LIN {X 0,Y 453.144,Z 723.625,A -85,B 0,C 180,E1 16875.324,E2 16875.324} C_VEL
LIN {X 0,Y 454.014,Z 710.614,A -85,B 0,C 180,E1 16875.765,E2 16875.765} C_VEL
LIN {X 0,Y 429.058,Z 654.338,A -85,B 0,C 180,E1 16879.298,E2 16879.298} C_VEL
LIN {X 0,Y 404.681,Z 601.31,A -85,B 0,C 180,E1 16882.971,E2 16882.971} C_VEL
LIN {X 0,Y 404.836,Z 601.31,A -85,B 0,C 180,E1 16889.422,E2 16889.422} C_VEL
LIN {X 0,Y 405.105,Z 601.31,A -85,B 0,C 180,E1 16895.708,E2 16895.708} C_VEL
LIN {X 0,Y 405.45,Z 601.31,A -85,B 0,C 180,E1 16902.605,E2 16902.605} C_VEL
LIN {X 0,Y 405.795,Z 601.31,A -85,B 0,C 180,E1 16909.24,E2 16909.24} C_VEL
LIN {X 0,Y 406.34,Z 601.31,A -85,B 0,C 180,E1 16915.721,E2 16915.721} C_VEL
LIN {X 0,Y 406.534,Z 601.31,A -85,B 0,C 180,E1 16922.133,E2 16922.133} C_VEL
LIN {X 0,Y 405.998,Z 601.31,A -85,B 0,C 180,E1 16928.581,E2 16928.581} C_VEL
LIN {X 0,Y 405.598,Z 601.31,A -85,B 0,C 180,E1 16935.153,E2 16935.153} C_VEL
LIN {X 0,Y 405.276,Z 601.31,A -85,B 0,C 180,E1 16941.947,E2 16941.947} C_VEL
LIN {X 0,Y 404.862,Z 601.31,A -85,B 0,C 180,E1 16949.103,E2 16949.103} C_VEL
LIN {X 0,Y 404.667,Z 601.31,A -85,B 0,C 180,E1 16954.527,E2 16954.527} C_VEL
LIN {X 0,Y 404.635,Z 601.31,A -85,B 0,C 180,E1 16961.494,E2 16961.494} C_VEL
LIN {X 0,Y 404.616,Z 601.411,A -85,B 0,C 180,E1 16963.759,E2 16963.759} C_VEL
LIN {X 0,Y 407.142,Z 607.04,A -85,B 0,C 180,E1 16964.41,E2 16964.41} C_VEL
LIN {X 0,Y 426.451,Z 643.441,A -85,B 0,C 180,E1 16968.623,E2 16968.623} C_VEL
LIN {X 0,Y 441.542,Z 679.841,A -85,B 0,C 180,E1 16971.916,E2 16971.916} C_VEL
LIN {X 0,Y 445.49,Z 694.589,A -85,B 0,C 180,E1 16973.129,E2 16973.129} C_VEL
LIN {X 0,Y 440.363,Z 731.801,A -85,B 0,C 180,E1 16975.298,E2 16975.298} C_VEL
LIN {X 0,Y 433.881,Z 767.453,A -85,B 0,C 180,E1 16978.257,E2 16978.257} C_VEL
LIN {X 0,Y 426.951,Z 799.424,A -85,B 0,C 180,E1 16981.945,E2 16981.945} C_VEL
LIN {X 0,Y 420.677,Z 825.936,A -85,B 0,C 180,E1 16986.09,E2 16986.09} C_VEL
LIN {X 0,Y 415.363,Z 848.097,A -85,B 0,C 180,E1 16990.828,E2 16990.828} C_VEL
LIN {X 0,Y 411.855,Z 864.058,A -85,B 0,C 180,E1 16995.615,E2 16995.615} C_VEL
LIN {X 0,Y 409.78,Z 874.937,A -85,B 0,C 180,E1 17000.416,E2 17000.416} C_VEL
LIN {X 0,Y 408.702,Z 881.698,A -85,B 0,C 180,E1 17005.742,E2 17005.742} C_VEL
LIN {X 0,Y 408.585,Z 883.379,A -85,B 0,C 180,E1 17009.994,E2 17009.994} C_VEL
LIN {X 0,Y 408.851,Z 880.711,A -85,B 0,C 180,E1 17015.31,E2 17015.31} C_VEL
LIN {X 0,Y 410.092,Z 872.747,A -85,B 0,C 180,E1 17020.64,E2 17020.64} C_VEL
LIN {X 0,Y 412.907,Z 859.065,A -85,B 0,C 180,E1 17025.969,E2 17025.969} C_VEL
LIN {X 0,Y 417.3,Z 839.904,A -85,B 0,C 180,E1 17031.006,E2 17031.006} C_VEL
LIN {X 0,Y 423.261,Z 814.998,A -85,B 0,C 180,E1 17035.669,E2 17035.669} C_VEL
LIN {X 0,Y 430.079,Z 785.455,A -85,B 0,C 180,E1 17039.706,E2 17039.706} C_VEL
LIN {X 0,Y 436.704,Z 752.798,A -85,B 0,C 180,E1 17042.97,E2 17042.97} C_VEL
LIN {X 0,Y 442.585,Z 716.698,A -85,B 0,C 180,E1 17045.585,E2 17045.585} C_VEL
LIN {X 0,Y 445.078,Z 692.222,A -85,B 0,C 180,E1 17046.937,E2 17046.937} C_VEL
LIN {X 0,Y 433.84,Z 659.714,A -85,B 0,C 180,E1 17049.714,E2 17049.714} C_VEL
LIN {X 0,Y 416.42,Z 623.579,A -85,B 0,C 180,E1 17053.415,E2 17053.415} C_VEL
LIN {X 0,Y 404.643,Z 601.978,A -85,B 0,C 180,E1 17056.084,E2 17056.084} C_VEL
LIN {X 0,Y 404.565,Z 601.31,A -85,B 0,C 180,E1 17061.851,E2 17061.851} C_VEL
LIN {X 0,Y 404.943,Z 601.976,A -85,B 0,C 180,E1 17068.085,E2 17068.085} C_VEL
LIN {X 0,Y 427.922,Z 668.698,A -85,B 0,C 180,E1 17071.46,E2 17071.46} C_VEL
LIN {X 0,Y 428.67,Z 678.715,A -85,B 0,C 180,E1 17071.781,E2 17071.781} C_VEL
LIN {X 0,Y 425.713,Z 719.893,A -85,B 0,C 180,E1 17073.236,E2 17073.236} C_VEL
LIN {X 0,Y 421.872,Z 759.16,A -85,B 0,C 180,E1 17075.471,E2 17075.471} C_VEL
LIN {X 0,Y 417.99,Z 794.434,A -85,B 0,C 180,E1 17078.39,E2 17078.39} C_VEL
LIN {X 0,Y 414.582,Z 824.543,A -85,B 0,C 180,E1 17081.831,E2 17081.831} C_VEL
LIN {X 0,Y 411.814,Z 848.973,A -85,B 0,C 180,E1 17085.626,E2 17085.626} C_VEL
LIN {X 0,Y 410.114,Z 868.93,A -85,B 0,C 180,E1 17089.898,E2 17089.898} C_VEL
LIN {X 0,Y 409.272,Z 882.602,A -85,B 0,C 180,E1 17094.161,E2 17094.161} C_VEL
LIN {X 0,Y 409.19,Z 891.235,A -85,B 0,C 180,E1 17098.574,E2 17098.574} C_VEL
LIN {X 0,Y 409.569,Z 894.347,A -85,B 0,C 180,E1 17102.122,E2 17102.122} C_VEL
LIN {X 0,Y 411.139,Z 893.587,A -85,B 0,C 180,E1 17106.349,E2 17106.349} C_VEL
LIN {X 0,Y 413.508,Z 887.959,A -85,B 0,C 180,E1 17110.557,E2 17110.557} C_VEL
LIN {X 0,Y 417.618,Z 875.892,A -85,B 0,C 180,E1 17115.115,E2 17115.115} C_VEL
LIN {X 0,Y 422.993,Z 858.13,A -85,B 0,C 180,E1 17119.349,E2 17119.349} C_VEL
LIN {X 0,Y 430.431,Z 833.334,A -85,B 0,C 180,E1 17123.442,E2 17123.442} C_VEL
LIN {X 0,Y 439.545,Z 802.14,A -85,B 0,C 180,E1 17127.174,E2 17127.174} C_VEL
LIN {X 0,Y 450.951,Z 763.363,A -85,B 0,C 180,E1 17130.54,E2 17130.54} C_VEL
LIN {X 0,Y 462.959,Z 721.781,A -85,B 0,C 180,E1 17133.048,E2 17133.048} C_VEL
LIN {X 0,Y 469.674,Z 695.489,A -85,B 0,C 180,E1 17134.267,E2 17134.267} C_VEL
LIN {X 0,Y 469.832,Z 688.161,A -85,B 0,C 180,E1 17136.141,E2 17136.141} C_VEL
LIN {X 0,Y 470.531,Z 686.318,A -85,B 0,C 180,E1 17137.657,E2 17137.657} C_VEL
LIN {X 0,Y 471.824,Z 691.946,A -85,B 0,C 180,E1 17139.617,E2 17139.617} C_VEL
LIN {X 0,Y 472.889,Z 702.024,A -85,B 0,C 180,E1 17141.096,E2 17141.096} C_VEL
LIN {X 0,Y 472.481,Z 713.92,A -85,B 0,C 180,E1 17142.03,E2 17142.03} C_VEL
LIN {X 0,Y 462.296,Z 759.297,A -85,B 0,C 180,E1 17143.95,E2 17143.95} C_VEL
LIN {X 0,Y 450.752,Z 803.897,A -85,B 0,C 180,E1 17146.773,E2 17146.773} C_VEL
LIN {X 0,Y 438.988,Z 845.741,A -85,B 0,C 180,E1 17150.484,E2 17150.484} C_VEL
LIN {X 0,Y 428.197,Z 882.986,A -85,B 0,C 180,E1 17154.933,E2 17154.933} C_VEL
LIN {X 0,Y 419.612,Z 914.659,A -85,B 0,C 180,E1 17159.961,E2 17159.961} C_VEL
LIN {X 0,Y 413.13,Z 941.761,A -85,B 0,C 180,E1 17165.638,E2 17165.638} C_VEL
LIN {X 0,Y 409.271,Z 963.039,A -85,B 0,C 180,E1 17171.664,E2 17171.664} C_VEL
LIN {X 0,Y 407.76,Z 977.862,A -85,B 0,C 180,E1 17177.669,E2 17177.669} C_VEL
LIN {X 0,Y 407.499,Z 985.661,A -85,B 0,C 180,E1 17182.528,E2 17182.528} C_VEL
LIN {X 0,Y 407.719,Z 989.763,A -85,B 0,C 180,E1 17187.876,E2 17187.876} C_VEL
LIN {X 0,Y 407.669,Z 989.715,A -85,B 0,C 180,E1 17192.136,E2 17192.136} C_VEL
LIN {X 0,Y 407.522,Z 985.383,A -85,B 0,C 180,E1 17197.483,E2 17197.483} C_VEL
LIN {X 0,Y 407.925,Z 976.144,A -85,B 0,C 180,E1 17202.883,E2 17202.883} C_VEL
LIN {X 0,Y 409.066,Z 963.513,A -85,B 0,C 180,E1 17207.72,E2 17207.72} C_VEL
LIN {X 0,Y 406.112,Z 956.241,A -85,B 0,C 180,E1 17209.923,E2 17209.923} C_VEL
LIN {X 0,Y 403.464,Z 948.232,A -85,B 0,C 180,E1 17212.111,E2 17212.111} C_VEL
LIN {X 0,Y 408.092,Z 924.272,A -85,B 0,C 180,E1 17217.467,E2 17217.467} C_VEL
LIN {X 0,Y 414.359,Z 895.799,A -85,B 0,C 180,E1 17222.261,E2 17222.261} C_VEL
LIN {X 0,Y 421.833,Z 862.647,A -85,B 0,C 180,E1 17226.508,E2 17226.508} C_VEL
LIN {X 0,Y 430.114,Z 823.849,A -85,B 0,C 180,E1 17230.223,E2 17230.223} C_VEL
LIN {X 0,Y 437.983,Z 781.87,A -85,B 0,C 180,E1 17233.15,E2 17233.15} C_VEL
LIN {X 0,Y 444.627,Z 738.33,A -85,B 0,C 180,E1 17235.268,E2 17235.268} C_VEL
LIN {X 0,Y 446.908,Z 712.636,A -85,B 0,C 180,E1 17236.208,E2 17236.208} C_VEL
LIN {X 0,Y 424.33,Z 661.374,A -85,B 0,C 180,E1 17239.508,E2 17239.508} C_VEL
LIN {X 0,Y 396.721,Z 601.31,A -85,B 0,C 180,E1 17243.82,E2 17243.82} C_VEL
LIN {X 0,Y 396.924,Z 601.31,A -85,B 0,C 180,E1 17250.251,E2 17250.251} C_VEL
LIN {X 0,Y 397.264,Z 601.31,A -85,B 0,C 180,E1 17257.581,E2 17257.581} C_VEL
LIN {X 0,Y 397.599,Z 601.31,A -85,B 0,C 180,E1 17264.529,E2 17264.529} C_VEL
LIN {X 0,Y 398.087,Z 601.31,A -85,B 0,C 180,E1 17271.778,E2 17271.778} C_VEL
LIN {X 0,Y 398.566,Z 601.31,A -85,B 0,C 180,E1 17277.819,E2 17277.819} C_VEL
LIN {X 0,Y 398.622,Z 601.31,A -85,B 0,C 180,E1 17282.175,E2 17282.175} C_VEL
LIN {X 0,Y 398.065,Z 601.31,A -85,B 0,C 180,E1 17288.753,E2 17288.753} C_VEL
LIN {X 0,Y 397.646,Z 601.31,A -85,B 0,C 180,E1 17295.464,E2 17295.464} C_VEL
LIN {X 0,Y 397.287,Z 601.31,A -85,B 0,C 180,E1 17302.412,E2 17302.412} C_VEL
LIN {X 0,Y 396.937,Z 601.31,A -85,B 0,C 180,E1 17309.741,E2 17309.741} C_VEL
LIN {X 0,Y 396.708,Z 601.31,A -85,B 0,C 180,E1 17316.66,E2 17316.66} C_VEL
LIN {X 0,Y 396.735,Z 601.61,A -85,B 0,C 180,E1 17322.493,E2 17322.493} C_VEL
LIN {X 0,Y 399.282,Z 607.13,A -85,B 0,C 180,E1 17323.171,E2 17323.171} C_VEL
LIN {X 0,Y 417.822,Z 641.308,A -85,B 0,C 180,E1 17327.427,E2 17327.427} C_VEL
LIN {X 0,Y 433.732,Z 678.097,A -85,B 0,C 180,E1 17330.964,E2 17330.964} C_VEL
LIN {X 0,Y 439.018,Z 697.43,A -85,B 0,C 180,E1 17332.614,E2 17332.614} C_VEL
LIN {X 0,Y 433.748,Z 733.916,A -85,B 0,C 180,E1 17334.796,E2 17334.796} C_VEL
LIN {X 0,Y 426.94,Z 769.727,A -85,B 0,C 180,E1 17337.829,E2 17337.829} C_VEL
LIN {X 0,Y 420.013,Z 800.415,A -85,B 0,C 180,E1 17341.439,E2 17341.439} C_VEL
LIN {X 0,Y 413.497,Z 826.928,A -85,B 0,C 180,E1 17345.648,E2 17345.648} C_VEL
LIN {X 0,Y 407.947,Z 849.099,A -85,B 0,C 180,E1 17350.465,E2 17350.465} C_VEL
LIN {X 0,Y 404.23,Z 865.06,A -85,B 0,C 180,E1 17355.338,E2 17355.338} C_VEL
LIN {X 0,Y 402.037,Z 875.93,A -85,B 0,C 180,E1 17360.23,E2 17360.23} C_VEL
LIN {X 0,Y 400.887,Z 882.687,A -85,B 0,C 180,E1 17365.659,E2 17365.659} C_VEL
LIN {X 0,Y 400.763,Z 884.365,A -85,B 0,C 180,E1 17369.994,E2 17369.994} C_VEL
LIN {X 0,Y 401.035,Z 881.701,A -85,B 0,C 180,E1 17375.414,E2 17375.414} C_VEL
LIN {X 0,Y 402.381,Z 873.742,A -85,B 0,C 180,E1 17380.846,E2 17380.846} C_VEL
LIN {X 0,Y 405.349,Z 860.066,A -85,B 0,C 180,E1 17386.275,E2 17386.275} C_VEL
LIN {X 0,Y 409.947,Z 840.904,A -85,B 0,C 180,E1 17391.401,E2 17391.401} C_VEL
LIN {X 0,Y 416.115,Z 816.225,A -85,B 0,C 180,E1 17396.102,E2 17396.102} C_VEL
LIN {X 0,Y 422.995,Z 787.652,A -85,B 0,C 180,E1 17400.092,E2 17400.092} C_VEL
LIN {X 0,Y 429.834,Z 755.218,A -85,B 0,C 180,E1 17403.415,E2 17403.415} C_VEL
LIN {X 0,Y 435.998,Z 719.092,A -85,B 0,C 180,E1 17406.095,E2 17406.095} C_VEL
LIN {X 0,Y 438.752,Z 695.217,A -85,B 0,C 180,E1 17407.432,E2 17407.432} C_VEL
LIN {X 0,Y 428.14,Z 663.804,A -85,B 0,C 180,E1 17410.203,E2 17410.203} C_VEL
LIN {X 0,Y 411.375,Z 628.716,A -85,B 0,C 180,E1 17413.89,E2 17413.89} C_VEL
LIN {X 0,Y 396.772,Z 602.597,A -85,B 0,C 180,E1 17417.323,E2 17417.323} C_VEL
LIN {X 0,Y 396.68,Z 601.31,A -85,B 0,C 180,E1 17417.552,E2 17417.552} C_VEL
LIN {X 0,Y 396.704,Z 601.31,A -85,B 0,C 180,E1 17425.058,E2 17425.058} C_VEL
LIN {X 0,Y 396.951,Z 601.31,A -85,B 0,C 180,E1 17427.466,E2 17427.466} C_VEL
LIN {X 0,Y 420.826,Z 670.997,A -85,B 0,C 180,E1 17431.112,E2 17431.112} C_VEL
LIN {X 0,Y 420.941,Z 686.929,A -85,B 0,C 180,E1 17431.596,E2 17431.596} C_VEL
LIN {X 0,Y 417.659,Z 727.911,A -85,B 0,C 180,E1 17433.231,E2 17433.231} C_VEL
LIN {X 0,Y 413.648,Z 766.912,A -85,B 0,C 180,E1 17435.672,E2 17435.672} C_VEL
LIN {X 0,Y 409.558,Z 802.307,A -85,B 0,C 180,E1 17438.864,E2 17438.864} C_VEL
LIN {X 0,Y 406.016,Z 832.346,A -85,B 0,C 180,E1 17442.636,E2 17442.636} C_VEL
LIN {X 0,Y 403.418,Z 856.03,A -85,B 0,C 180,E1 17446.706,E2 17446.706} C_VEL
LIN {X 0,Y 401.855,Z 875.142,A -85,B 0,C 180,E1 17451.33,E2 17451.33} C_VEL
LIN {X 0,Y 401.38,Z 887.036,A -85,B 0,C 180,E1 17455.674,E2 17455.674} C_VEL
LIN {X 0,Y 401.482,Z 893.849,A -85,B 0,C 180,E1 17460.003,E2 17460.003} C_VEL
LIN {X 0,Y 402.47,Z 895.827,A -85,B 0,C 180,E1 17464.32,E2 17464.32} C_VEL
LIN {X 0,Y 404.529,Z 892.945,A -85,B 0,C 180,E1 17468.618,E2 17468.618} C_VEL
LIN {X 0,Y 408.246,Z 883.721,A -85,B 0,C 180,E1 17473.413,E2 17473.413} C_VEL
LIN {X 0,Y 412.904,Z 870.089,A -85,B 0,C 180,E1 17477.566,E2 17477.566} C_VEL
LIN {X 0,Y 419.579,Z 850.051,A -85,B 0,C 180,E1 17481.723,E2 17481.723} C_VEL
LIN {X 0,Y 428.729,Z 821.406,A -85,B 0,C 180,E1 17485.932,E2 17485.932} C_VEL
LIN {X 0,Y 440.153,Z 786.19,A -85,B 0,C 180,E1 17489.656,E2 17489.656} C_VEL
LIN {X 0,Y 452.998,Z 746.965,A -85,B 0,C 180,E1 17492.635,E2 17492.635} C_VEL
LIN {X 0,Y 465.569,Z 706.07,A -85,B 0,C 180,E1 17494.732,E2 17494.732} C_VEL
LIN {X 0,Y 467.104,Z 699.977,A -85,B 0,C 180,E1 17495.095,E2 17495.095} C_VEL
LIN {X 0,Y 467.92,Z 694.621,A -85,B 0,C 180,E1 17496.923,E2 17496.923} C_VEL
LIN {X 0,Y 468.515,Z 695.099,A -85,B 0,C 180,E1 17498.092,E2 17498.092} C_VEL
LIN {X 0,Y 469.391,Z 701.137,A -85,B 0,C 180,E1 17499.712,E2 17499.712} C_VEL
LIN {X 0,Y 469.233,Z 712.69,A -85,B 0,C 180,E1 17500.993,E2 17500.993} C_VEL
LIN {X 0,Y 456.969,Z 763.857,A -85,B 0,C 180,E1 17503.339,E2 17503.339} C_VEL
LIN {X 0,Y 444.904,Z 806.362,A -85,B 0,C 180,E1 17506.155,E2 17506.155} C_VEL
LIN {X 0,Y 432.505,Z 847.465,A -85,B 0,C 180,E1 17509.936,E2 17509.936} C_VEL
LIN {X 0,Y 421.413,Z 883.423,A -85,B 0,C 180,E1 17514.373,E2 17514.373} C_VEL
LIN {X 0,Y 412.458,Z 914.186,A -85,B 0,C 180,E1 17519.385,E2 17519.385} C_VEL
LIN {X 0,Y 405.947,Z 939.975,A -85,B 0,C 180,E1 17524.883,E2 17524.883} C_VEL
LIN {X 0,Y 401.699,Z 961.213,A -85,B 0,C 180,E1 17530.941,E2 17530.941} C_VEL
LIN {X 0,Y 399.921,Z 977.012,A -85,B 0,C 180,E1 17537.423,E2 17537.423} C_VEL
LIN {X 0,Y 399.618,Z 984.745,A -85,B 0,C 180,E1 17542.38,E2 17542.38} C_VEL
LIN {X 0,Y 399.888,Z 988.813,A -85,B 0,C 180,E1 17547.834,E2 17547.834} C_VEL
LIN {X 0,Y 399.842,Z 988.709,A -85,B 0,C 180,E1 17552.178,E2 17552.178} C_VEL
LIN {X 0,Y 399.685,Z 984.293,A -85,B 0,C 180,E1 17557.631,E2 17557.631} C_VEL
LIN {X 0,Y 400.089,Z 974.873,A -85,B 0,C 180,E1 17563.14,E2 17563.14} C_VEL
LIN {X 0,Y 401.48,Z 960.573,A -85,B 0,C 180,E1 17568.582,E2 17568.582} C_VEL
LIN {X 0,Y 403.464,Z 948.232,A -85,B 0,C 180,E1 17572.111,E2 17572.111} C_VEL
LIN {X 0,Y 401.121,Z 939.612,A -85,B 0,C 180,E1 17574.259,E2 17574.259} C_VEL
LIN {X 0,Y 399.038,Z 930.299,A -85,B 0,C 180,E1 17576.378,E2 17576.378} C_VEL
LIN {X 0,Y 405.037,Z 903.022,A -85,B 0,C 180,E1 17581.397,E2 17581.397} C_VEL
LIN {X 0,Y 412.444,Z 871.136,A -85,B 0,C 180,E1 17585.845,E2 17585.845} C_VEL
LIN {X 0,Y 420.387,Z 835.553,A -85,B 0,C 180,E1 17589.607,E2 17589.607} C_VEL
LIN {X 0,Y 428.414,Z 796.139,A -85,B 0,C 180,E1 17592.707,E2 17592.707} C_VEL
LIN {X 0,Y 435.678,Z 753.012,A -85,B 0,C 180,E1 17595.129,E2 17595.129} C_VEL
LIN {X 0,Y 439.896,Z 715.013,A -85,B 0,C 180,E1 17596.636,E2 17596.636} C_VEL
LIN {X 0,Y 419.655,Z 668.36,A -85,B 0,C 180,E1 17599.719,E2 17599.719} C_VEL
LIN {X 0,Y 388.811,Z 601.31,A -85,B 0,C 180,E1 17604.558,E2 17604.558} C_VEL
LIN {X 0,Y 389.049,Z 601.31,A -85,B 0,C 180,E1 17612.14,E2 17612.14} C_VEL
LIN {X 0,Y 389.433,Z 601.31,A -85,B 0,C 180,E1 17619.504,E2 17619.504} C_VEL
LIN {X 0,Y 389.826,Z 601.31,A -85,B 0,C 180,E1 17626.514,E2 17626.514} C_VEL
LIN {X 0,Y 390.335,Z 601.31,A -85,B 0,C 180,E1 17633.311,E2 17633.311} C_VEL
LIN {X 0,Y 390.868,Z 601.31,A -85,B 0,C 180,E1 17639.997,E2 17639.997} C_VEL
LIN {X 0,Y 390.34,Z 601.31,A -85,B 0,C 180,E1 17646.683,E2 17646.683} C_VEL
LIN {X 0,Y 389.843,Z 601.31,A -85,B 0,C 180,E1 17653.643,E2 17653.643} C_VEL
LIN {X 0,Y 389.412,Z 601.31,A -85,B 0,C 180,E1 17660.941,E2 17660.941} C_VEL
LIN {X 0,Y 389.034,Z 601.31,A -85,B 0,C 180,E1 17667.854,E2 17667.854} C_VEL
LIN {X 0,Y 388.844,Z 601.31,A -85,B 0,C 180,E1 17675.074,E2 17675.074} C_VEL
LIN {X 0,Y 388.797,Z 601.546,A -85,B 0,C 180,E1 17681.118,E2 17681.118} C_VEL
LIN {X 0,Y 391.283,Z 607.066,A -85,B 0,C 180,E1 17681.818,E2 17681.818} C_VEL
LIN {X 0,Y 409.624,Z 639.903,A -85,B 0,C 180,E1 17686.242,E2 17686.242} C_VEL
LIN {X 0,Y 426.017,Z 676.952,A -85,B 0,C 180,E1 17690.025,E2 17690.025} C_VEL
LIN {X 0,Y 432.632,Z 699.526,A -85,B 0,C 180,E1 17692.046,E2 17692.046} C_VEL
LIN {X 0,Y 427.133,Z 736.226,A -85,B 0,C 180,E1 17694.293,E2 17694.293} C_VEL
LIN {X 0,Y 420.051,Z 771.896,A -85,B 0,C 180,E1 17697.381,E2 17697.381} C_VEL
LIN {X 0,Y 412.682,Z 803.295,A -85,B 0,C 180,E1 17701.184,E2 17701.184} C_VEL
LIN {X 0,Y 405.602,Z 830.769,A -85,B 0,C 180,E1 17705.731,E2 17705.731} C_VEL
LIN {X 0,Y 400.01,Z 852,A -85,B 0,C 180,E1 17710.601,E2 17710.601} C_VEL
LIN {X 0,Y 395.958,Z 868.944,A -85,B 0,C 180,E1 17716.156,E2 17716.156} C_VEL
LIN {X 0,Y 393.908,Z 878.753,A -85,B 0,C 180,E1 17721.143,E2 17721.143} C_VEL
LIN {X 0,Y 393.089,Z 883.674,A -85,B 0,C 180,E1 17725.572,E2 17725.572} C_VEL
LIN {X 0,Y 392.955,Z 885.35,A -85,B 0,C 180,E1 17729.994,E2 17729.994} C_VEL
LIN {X 0,Y 393.241,Z 882.688,A -85,B 0,C 180,E1 17735.522,E2 17735.522} C_VEL
LIN {X 0,Y 394.681,Z 874.735,A -85,B 0,C 180,E1 17741.061,E2 17741.061} C_VEL
LIN {X 0,Y 397.776,Z 861.078,A -85,B 0,C 180,E1 17746.594,E2 17746.594} C_VEL
LIN {X 0,Y 402.63,Z 841.907,A -85,B 0,C 180,E1 17751.809,E2 17751.809} C_VEL
LIN {X 0,Y 409.074,Z 817.24,A -85,B 0,C 180,E1 17756.585,E2 17756.585} C_VEL
LIN {X 0,Y 416.212,Z 788.636,A -85,B 0,C 180,E1 17760.635,E2 17760.635} C_VEL
LIN {X 0,Y 423.326,Z 756.172,A -85,B 0,C 180,E1 17763.998,E2 17763.998} C_VEL
LIN {X 0,Y 429.751,Z 719.457,A -85,B 0,C 180,E1 17766.741,E2 17766.741} C_VEL
LIN {X 0,Y 432.249,Z 697.341,A -85,B 0,C 180,E1 17768.015,E2 17768.015} C_VEL
LIN {X 0,Y 421.482,Z 665.442,A -85,B 0,C 180,E1 17770.935,E2 17770.935} C_VEL
LIN {X 0,Y 404.201,Z 629.523,A -85,B 0,C 180,E1 17774.901,E2 17774.901} C_VEL
LIN {X 0,Y 390.003,Z 605.572,A -85,B 0,C 180,E1 17778.345,E2 17778.345} C_VEL
LIN {X 0,Y 388.737,Z 601.31,A -85,B 0,C 180,E1 17778.808,E2 17778.808} C_VEL
LIN {X 0,Y 388.985,Z 601.31,A -85,B 0,C 180,E1 17786.898,E2 17786.898} C_VEL
LIN {X 0,Y 412.526,Z 669.642,A -85,B 0,C 180,E1 17790.575,E2 17790.575} C_VEL
LIN {X 0,Y 414.213,Z 677.972,A -85,B 0,C 180,E1 17790.919,E2 17790.919} C_VEL
LIN {X 0,Y 411.094,Z 719.632,A -85,B 0,C 180,E1 17792.43,E2 17792.43} C_VEL
LIN {X 0,Y 407.087,Z 758.185,A -85,B 0,C 180,E1 17794.666,E2 17794.666} C_VEL
LIN {X 0,Y 402.859,Z 794.573,A -85,B 0,C 180,E1 17797.74,E2 17797.74} C_VEL
LIN {X 0,Y 399.041,Z 826.575,A -85,B 0,C 180,E1 17801.517,E2 17801.517} C_VEL
LIN {X 0,Y 396.091,Z 851.835,A -85,B 0,C 180,E1 17805.608,E2 17805.608} C_VEL
LIN {X 0,Y 394.356,Z 871.599,A -85,B 0,C 180,E1 17810.048,E2 17810.048} C_VEL
LIN {X 0,Y 393.543,Z 885.173,A -85,B 0,C 180,E1 17814.48,E2 17814.48} C_VEL
LIN {X 0,Y 393.556,Z 893.492,A -85,B 0,C 180,E1 17818.9,E2 17818.9} C_VEL
LIN {X 0,Y 393.94,Z 896.554,A -85,B 0,C 180,E1 17822.207,E2 17822.207} C_VEL
LIN {X 0,Y 395.687,Z 896.345,A -85,B 0,C 180,E1 17826.598,E2 17826.598} C_VEL
LIN {X 0,Y 398.826,Z 890.34,A -85,B 0,C 180,E1 17831.505,E2 17831.505} C_VEL
LIN {X 0,Y 403.433,Z 878.844,A -85,B 0,C 180,E1 17836.082,E2 17836.082} C_VEL
LIN {X 0,Y 409.889,Z 861.011,A -85,B 0,C 180,E1 17840.558,E2 17840.558} C_VEL
LIN {X 0,Y 418.813,Z 835.899,A -85,B 0,C 180,E1 17844.927,E2 17844.927} C_VEL
LIN {X 0,Y 430.242,Z 803.687,A -85,B 0,C 180,E1 17848.959,E2 17848.959} C_VEL
LIN {X 0,Y 444.537,Z 764.527,A -85,B 0,C 180,E1 17852.464,E2 17852.464} C_VEL
LIN {X 0,Y 458.962,Z 723.662,A -85,B 0,C 180,E1 17854.961,E2 17854.961} C_VEL
LIN {X 0,Y 464.376,Z 706.896,A -85,B 0,C 180,E1 17855.698,E2 17855.698} C_VEL
LIN {X 0,Y 465.29,Z 703.344,A -85,B 0,C 180,E1 17856.422,E2 17856.422} C_VEL
LIN {X 0,Y 466.118,Z 702.017,A -85,B 0,C 180,E1 17857.685,E2 17857.685} C_VEL
LIN {X 0,Y 466.541,Z 706.311,A -85,B 0,C 180,E1 17859.045,E2 17859.045} C_VEL
LIN {X 0,Y 465.817,Z 716.907,A -85,B 0,C 180,E1 17860.288,E2 17860.288} C_VEL
LIN {X 0,Y 453.031,Z 764.068,A -85,B 0,C 180,E1 17862.453,E2 17862.453} C_VEL
LIN {X 0,Y 439.872,Z 806.951,A -85,B 0,C 180,E1 17865.354,E2 17865.354} C_VEL
LIN {X 0,Y 426.456,Z 848.229,A -85,B 0,C 180,E1 17869.249,E2 17869.249} C_VEL
LIN {X 0,Y 414.912,Z 883.26,A -85,B 0,C 180,E1 17873.689,E2 17873.689} C_VEL
LIN {X 0,Y 404.968,Z 915.321,A -85,B 0,C 180,E1 17879.083,E2 17879.083} C_VEL
LIN {X 0,Y 397.951,Z 941.528,A -85,B 0,C 180,E1 17884.945,E2 17884.945} C_VEL
LIN {X 0,Y 393.692,Z 962.019,A -85,B 0,C 180,E1 17891.131,E2 17891.131} C_VEL
LIN {X 0,Y 392.052,Z 976.171,A -85,B 0,C 180,E1 17897.166,E2 17897.166} C_VEL
LIN {X 0,Y 391.746,Z 983.826,A -85,B 0,C 180,E1 17902.226,E2 17902.226} C_VEL
LIN {X 0,Y 392.031,Z 987.858,A -85,B 0,C 180,E1 17907.791,E2 17907.791} C_VEL
LIN {X 0,Y 391.995,Z 987.69,A -85,B 0,C 180,E1 17912.221,E2 17912.221} C_VEL
LIN {X 0,Y 391.843,Z 983.185,A -85,B 0,C 180,E1 17917.784,E2 17917.784} C_VEL
LIN {X 0,Y 392.272,Z 973.572,A -85,B 0,C 180,E1 17923.407,E2 17923.407} C_VEL
LIN {X 0,Y 393.735,Z 959.322,A -85,B 0,C 180,E1 17928.882,E2 17928.882} C_VEL
LIN {X 0,Y 397.604,Z 937.515,A -85,B 0,C 180,E1 17934.79,E2 17934.79} C_VEL
LIN {X 0,Y 399.038,Z 930.299,A -85,B 0,C 180,E1 17936.378,E2 17936.378} C_VEL
LIN {X 0,Y 397.383,Z 920.418,A -85,B 0,C 180,E1 17938.443,E2 17938.443} C_VEL
LIN {X 0,Y 395.78,Z 909.888,A -85,B 0,C 180,E1 17940.468,E2 17940.468} C_VEL
LIN {X 0,Y 403.531,Z 877.009,A -85,B 0,C 180,E1 17945.434,E2 17945.434} C_VEL
LIN {X 0,Y 412.134,Z 839.758,A -85,B 0,C 180,E1 17949.613,E2 17949.613} C_VEL
LIN {X 0,Y 420.912,Z 797.997,A -85,B 0,C 180,E1 17953.034,E2 17953.034} C_VEL
LIN {X 0,Y 428.714,Z 752.963,A -85,B 0,C 180,E1 17955.622,E2 17955.622} C_VEL
LIN {X 0,Y 432.857,Z 717.222,A -85,B 0,C 180,E1 17957.076,E2 17957.076} C_VEL
LIN {X 0,Y 413.269,Z 671.841,A -85,B 0,C 180,E1 17960.16,E2 17960.16} C_VEL
LIN {X 0,Y 380.863,Z 601.31,A -85,B 0,C 180,E1 17965.421,E2 17965.421} C_VEL
LIN {X 0,Y 381.041,Z 601.31,A -85,B 0,C 180,E1 17971.502,E2 17971.502} C_VEL
LIN {X 0,Y 381.511,Z 601.31,A -85,B 0,C 180,E1 17979.058,E2 17979.058} C_VEL
LIN {X 0,Y 381.888,Z 601.31,A -85,B 0,C 180,E1 17986.228,E2 17986.228} C_VEL
LIN {X 0,Y 382.401,Z 601.31,A -85,B 0,C 180,E1 17993.172,E2 17993.172} C_VEL
LIN {X 0,Y 382.965,Z 601.31,A -85,B 0,C 180,E1 17999.997,E2 17999.997} C_VEL
LIN {X 0,Y 382.406,Z 601.31,A -85,B 0,C 180,E1 18006.822,E2 18006.822} C_VEL
LIN {X 0,Y 381.938,Z 601.31,A -85,B 0,C 180,E1 18013.764,E2 18013.764} C_VEL
LIN {X 0,Y 381.524,Z 601.31,A -85,B 0,C 180,E1 18020.935,E2 18020.935} C_VEL
LIN {X 0,Y 381.034,Z 601.31,A -85,B 0,C 180,E1 18028.492,E2 18028.492} C_VEL
LIN {X 0,Y 380.917,Z 601.31,A -85,B 0,C 180,E1 18033.829,E2 18033.829} C_VEL
LIN {X 0,Y 380.9,Z 601.994,A -85,B 0,C 180,E1 18039.667,E2 18039.667} C_VEL
LIN {X 0,Y 383.969,Z 607.562,A -85,B 0,C 180,E1 18040.529,E2 18040.529} C_VEL
LIN {X 0,Y 403.157,Z 642.248,A -85,B 0,C 180,E1 18045.418,E2 18045.418} C_VEL
LIN {X 0,Y 419.103,Z 677.789,A -85,B 0,C 180,E1 18049.233,E2 18049.233} C_VEL
LIN {X 0,Y 426.223,Z 702.315,A -85,B 0,C 180,E1 18051.502,E2 18051.502} C_VEL
LIN {X 0,Y 420.319,Z 739.659,A -85,B 0,C 180,E1 18053.853,E2 18053.853} C_VEL
LIN {X 0,Y 413.263,Z 773.734,A -85,B 0,C 180,E1 18056.886,E2 18056.886} C_VEL
LIN {X 0,Y 405.796,Z 804.297,A -85,B 0,C 180,E1 18060.648,E2 18060.648} C_VEL
LIN {X 0,Y 398.839,Z 830.381,A -85,B 0,C 180,E1 18064.992,E2 18064.992} C_VEL
LIN {X 0,Y 392.726,Z 852.532,A -85,B 0,C 180,E1 18070.089,E2 18070.089} C_VEL
LIN {X 0,Y 388.658,Z 868.499,A -85,B 0,C 180,E1 18075.315,E2 18075.315} C_VEL
LIN {X 0,Y 386.142,Z 879.744,A -85,B 0,C 180,E1 18080.963,E2 18080.963} C_VEL
LIN {X 0,Y 385.275,Z 884.662,A -85,B 0,C 180,E1 18085.482,E2 18085.482} C_VEL
LIN {X 0,Y 385.134,Z 886.336,A -85,B 0,C 180,E1 18089.994,E2 18089.994} C_VEL
LIN {X 0,Y 385.427,Z 883.679,A -85,B 0,C 180,E1 18095.634,E2 18095.634} C_VEL
LIN {X 0,Y 386.967,Z 875.731,A -85,B 0,C 180,E1 18101.284,E2 18101.284} C_VEL
LIN {X 0,Y 390.229,Z 862.086,A -85,B 0,C 180,E1 18106.924,E2 18106.924} C_VEL
LIN {X 0,Y 395.343,Z 842.906,A -85,B 0,C 180,E1 18112.233,E2 18112.233} C_VEL
LIN {X 0,Y 401.776,Z 819.341,A -85,B 0,C 180,E1 18116.901,E2 18116.901} C_VEL
LIN {X 0,Y 409.471,Z 789.626,A -85,B 0,C 180,E1 18121.195,E2 18121.195} C_VEL
LIN {X 0,Y 416.86,Z 757.165,A -85,B 0,C 180,E1 18124.6,E2 18124.6} C_VEL
LIN {X 0,Y 423.499,Z 720.346,A -85,B 0,C 180,E1 18127.374,E2 18127.374} C_VEL
LIN {X 0,Y 426.031,Z 700.361,A -85,B 0,C 180,E1 18128.535,E2 18128.535} C_VEL
LIN {X 0,Y 415.448,Z 668.603,A -85,B 0,C 180,E1 18131.548,E2 18131.548} C_VEL
LIN {X 0,Y 399.082,Z 634.376,A -85,B 0,C 180,E1 18135.452,E2 18135.452} C_VEL
LIN {X 0,Y 382.861,Z 606.575,A -85,B 0,C 180,E1 18139.594,E2 18139.594} C_VEL
LIN {X 0,Y 380.84,Z 601.31,A -85,B 0,C 180,E1 18140.269,E2 18140.269} C_VEL
LIN {X 0,Y 380.999,Z 601.375,A -85,B 0,C 180,E1 18146.292,E2 18146.292} C_VEL
LIN {X 0,Y 404.703,Z 669.495,A -85,B 0,C 180,E1 18150.087,E2 18150.087} C_VEL
LIN {X 0,Y 406.882,Z 679.535,A -85,B 0,C 180,E1 18150.525,E2 18150.525} C_VEL
LIN {X 0,Y 403.588,Z 720.868,A -85,B 0,C 180,E1 18152.083,E2 18152.083} C_VEL
LIN {X 0,Y 399.409,Z 760.224,A -85,B 0,C 180,E1 18154.445,E2 18154.445} C_VEL
LIN {X 0,Y 395.094,Z 796.523,A -85,B 0,C 180,E1 18157.606,E2 18157.606} C_VEL
LIN {X 0,Y 391.231,Z 827.882,A -85,B 0,C 180,E1 18161.398,E2 18161.398} C_VEL
LIN {X 0,Y 388.21,Z 853.229,A -85,B 0,C 180,E1 18165.598,E2 18165.598} C_VEL
LIN {X 0,Y 386.452,Z 872.892,A -85,B 0,C 180,E1 18170.128,E2 18170.128} C_VEL
LIN {X 0,Y 385.66,Z 887.137,A -85,B 0,C 180,E1 18174.932,E2 18174.932} C_VEL
LIN {X 0,Y 385.726,Z 894.337,A -85,B 0,C 180,E1 18178.878,E2 18178.878} C_VEL
LIN {X 0,Y 386.126,Z 897.642,A -85,B 0,C 180,E1 18182.251,E2 18182.251} C_VEL
LIN {X 0,Y 387.97,Z 897.729,A -85,B 0,C 180,E1 18186.73,E2 18186.73} C_VEL
LIN {X 0,Y 390.802,Z 893.049,A -85,B 0,C 180,E1 18191.178,E2 18191.178} C_VEL
LIN {X 0,Y 395.176,Z 883.402,A -85,B 0,C 180,E1 18195.568,E2 18195.568} C_VEL
LIN {X 0,Y 401.588,Z 867.375,A -85,B 0,C 180,E1 18200.137,E2 18200.137} C_VEL
LIN {X 0,Y 410.828,Z 843.843,A -85,B 0,C 180,E1 18204.687,E2 18204.687} C_VEL
LIN {X 0,Y 422.716,Z 813.226,A -85,B 0,C 180,E1 18208.937,E2 18208.937} C_VEL
LIN {X 0,Y 437.646,Z 776.296,A -85,B 0,C 180,E1 18212.597,E2 18212.597} C_VEL
LIN {X 0,Y 452.911,Z 738.111,A -85,B 0,C 180,E1 18215.241,E2 18215.241} C_VEL
LIN {X 0,Y 462.665,Z 711.247,A -85,B 0,C 180,E1 18216.54,E2 18216.54} C_VEL
LIN {X 0,Y 463.392,Z 709.586,A -85,B 0,C 180,E1 18217.207,E2 18217.207} C_VEL
LIN {X 0,Y 463.719,Z 711.742,A -85,B 0,C 180,E1 18218.37,E2 18218.37} C_VEL
LIN {X 0,Y 462.861,Z 719.733,A -85,B 0,C 180,E1 18219.444,E2 18219.444} C_VEL
LIN {X 0,Y 449.315,Z 764.923,A -85,B 0,C 180,E1 18221.567,E2 18221.567} C_VEL
LIN {X 0,Y 435.07,Z 807.689,A -85,B 0,C 180,E1 18224.53,E2 18224.53} C_VEL
LIN {X 0,Y 420.531,Z 849.248,A -85,B 0,C 180,E1 18228.55,E2 18228.55} C_VEL
LIN {X 0,Y 407.353,Z 886.643,A -85,B 0,C 180,E1 18233.485,E2 18233.485} C_VEL
LIN {X 0,Y 396.682,Z 919.305,A -85,B 0,C 180,E1 18239.34,E2 18239.34} C_VEL
LIN {X 0,Y 389.222,Z 945.494,A -85,B 0,C 180,E1 18245.665,E2 18245.665} C_VEL
LIN {X 0,Y 385.325,Z 965.301,A -85,B 0,C 180,E1 18252.263,E2 18252.263} C_VEL
LIN {X 0,Y 384.013,Z 978.238,A -85,B 0,C 180,E1 18258.628,E2 18258.628} C_VEL
LIN {X 0,Y 383.949,Z 984.065,A -85,B 0,C 180,E1 18263.207,E2 18263.207} C_VEL
LIN {X 0,Y 384.199,Z 986.9,A -85,B 0,C 180,E1 18267.746,E2 18267.746} C_VEL
LIN {X 0,Y 384.167,Z 986.659,A -85,B 0,C 180,E1 18272.267,E2 18272.267} C_VEL
LIN {X 0,Y 383.976,Z 982.054,A -85,B 0,C 180,E1 18277.945,E2 18277.945} C_VEL
LIN {X 0,Y 384.445,Z 972.243,A -85,B 0,C 180,E1 18283.685,E2 18283.685} C_VEL
LIN {X 0,Y 386.085,Z 957.46,A -85,B 0,C 180,E1 18289.36,E2 18289.36} C_VEL
LIN {X 0,Y 390.072,Z 935.637,A -85,B 0,C 180,E1 18295.302,E2 18295.302} C_VEL
LIN {X 0,Y 395.78,Z 909.888,A -85,B 0,C 180,E1 18300.468,E2 18300.468} C_VEL
LIN {X 0,Y 394.354,Z 898.826,A -85,B 0,C 180,E1 18302.436,E2 18302.436} C_VEL
LIN {X 0,Y 393.422,Z 887.17,A -85,B 0,C 180,E1 18304.338,E2 18304.338} C_VEL
LIN {X 0,Y 402.375,Z 850.213,A -85,B 0,C 180,E1 18308.939,E2 18308.939} C_VEL
LIN {X 0,Y 411.469,Z 809.362,A -85,B 0,C 180,E1 18312.65,E2 18312.65} C_VEL
LIN {X 0,Y 419.463,Z 766.309,A -85,B 0,C 180,E1 18315.45,E2 18315.45} C_VEL
LIN {X 0,Y 425.925,Z 721.543,A -85,B 0,C 180,E1 18317.424,E2 18317.424} C_VEL
LIN {X 0,Y 410.947,Z 684.418,A -85,B 0,C 180,E1 18319.996,E2 18319.996} C_VEL
LIN {X 0,Y 373,Z 601.31,A -85,B 0,C 180,E1 18326.225,E2 18326.225} C_VEL
LIN {X 0,Y 373.2,Z 601.31,A -85,B 0,C 180,E1 18333.477,E2 18333.477} C_VEL
LIN {X 0,Y 373.596,Z 601.31,A -85,B 0,C 180,E1 18338.896,E2 18338.896} C_VEL
LIN {X 0,Y 373.995,Z 601.31,A -85,B 0,C 180,E1 18346.519,E2 18346.519} C_VEL
LIN {X 0,Y 374.475,Z 601.31,A -85,B 0,C 180,E1 18353.026,E2 18353.026} C_VEL
LIN {X 0,Y 375.061,Z 601.31,A -85,B 0,C 180,E1 18359.997,E2 18359.997} C_VEL
LIN {X 0,Y 374.48,Z 601.31,A -85,B 0,C 180,E1 18366.968,E2 18366.968} C_VEL
LIN {X 0,Y 373.976,Z 601.31,A -85,B 0,C 180,E1 18374.063,E2 18374.063} C_VEL
LIN {X 0,Y 373.551,Z 601.31,A -85,B 0,C 180,E1 18381.403,E2 18381.403} C_VEL
LIN {X 0,Y 373.102,Z 601.31,A -85,B 0,C 180,E1 18389.155,E2 18389.155} C_VEL
LIN {X 0,Y 372.823,Z 601.31,A -85,B 0,C 180,E1 18395.616,E2 18395.616} C_VEL
LIN {X 0,Y 372.83,Z 601.581,A -85,B 0,C 180,E1 18398.022,E2 18398.022} C_VEL
LIN {X 0,Y 375.405,Z 607.076,A -85,B 0,C 180,E1 18398.846,E2 18398.846} C_VEL
LIN {X 0,Y 391.314,Z 634.167,A -85,B 0,C 180,E1 18403.175,E2 18403.175} C_VEL
LIN {X 0,Y 407.316,Z 666.879,A -85,B 0,C 180,E1 18407.187,E2 18407.187} C_VEL
LIN {X 0,Y 418.071,Z 696.264,A -85,B 0,C 180,E1 18410.145,E2 18410.145} C_VEL
LIN {X 0,Y 419.727,Z 705.916,A -85,B 0,C 180,E1 18410.986,E2 18410.986} C_VEL
LIN {X 0,Y 413.838,Z 741.512,A -85,B 0,C 180,E1 18413.283,E2 18413.283} C_VEL
LIN {X 0,Y 406.132,Z 777.11,A -85,B 0,C 180,E1 18416.544,E2 18416.544} C_VEL
LIN {X 0,Y 398.47,Z 807.17,A -85,B 0,C 180,E1 18420.367,E2 18420.367} C_VEL
LIN {X 0,Y 390.938,Z 834.044,A -85,B 0,C 180,E1 18425.044,E2 18425.044} C_VEL
LIN {X 0,Y 384.793,Z 855.443,A -85,B 0,C 180,E1 18430.229,E2 18430.229} C_VEL
LIN {X 0,Y 380.687,Z 870.935,A -85,B 0,C 180,E1 18435.589,E2 18435.589} C_VEL
LIN {X 0,Y 378.379,Z 880.736,A -85,B 0,C 180,E1 18440.776,E2 18440.776} C_VEL
LIN {X 0,Y 377.478,Z 885.65,A -85,B 0,C 180,E1 18445.389,E2 18445.389} C_VEL
LIN {X 0,Y 377.295,Z 887.324,A -85,B 0,C 180,E1 18449.994,E2 18449.994} C_VEL
LIN {X 0,Y 377.63,Z 884.669,A -85,B 0,C 180,E1 18455.751,E2 18455.751} C_VEL
LIN {X 0,Y 379.259,Z 876.732,A -85,B 0,C 180,E1 18461.516,E2 18461.516} C_VEL
LIN {X 0,Y 382.681,Z 863.098,A -85,B 0,C 180,E1 18467.268,E2 18467.268} C_VEL
LIN {X 0,Y 388.06,Z 843.918,A -85,B 0,C 180,E1 18472.673,E2 18472.673} C_VEL
LIN {X 0,Y 394.766,Z 820.354,A -85,B 0,C 180,E1 18477.418,E2 18477.418} C_VEL
LIN {X 0,Y 402.765,Z 790.621,A -85,B 0,C 180,E1 18481.774,E2 18481.774} C_VEL
LIN {X 0,Y 410.439,Z 758.143,A -85,B 0,C 180,E1 18485.22,E2 18485.22} C_VEL
LIN {X 0,Y 417.286,Z 721.237,A -85,B 0,C 180,E1 18488.028,E2 18488.028} C_VEL
LIN {X 0,Y 419.627,Z 702.543,A -85,B 0,C 180,E1 18489.148,E2 18489.148} C_VEL
LIN {X 0,Y 409.456,Z 671.742,A -85,B 0,C 180,E1 18492.178,E2 18492.178} C_VEL
LIN {X 0,Y 393.737,Z 638.684,A -85,B 0,C 180,E1 18496.077,E2 18496.077} C_VEL
LIN {X 0,Y 375.845,Z 607.491,A -85,B 0,C 180,E1 18500.907,E2 18500.907} C_VEL
LIN {X 0,Y 372.831,Z 602.234,A -85,B 0,C 180,E1 18501.812,E2 18501.812} C_VEL
LIN {X 0,Y 372.788,Z 601.31,A -85,B 0,C 180,E1 18502.447,E2 18502.447} C_VEL
LIN {X 0,Y 372.961,Z 601.31,A -85,B 0,C 180,E1 18505.65,E2 18505.65} C_VEL
LIN {X 0,Y 396.072,Z 667.209,A -85,B 0,C 180,E1 18509.477,E2 18509.477} C_VEL
LIN {X 0,Y 399.613,Z 679.843,A -85,B 0,C 180,E1 18510.095,E2 18510.095} C_VEL
LIN {X 0,Y 396.138,Z 722.214,A -85,B 0,C 180,E1 18511.738,E2 18511.738} C_VEL
LIN {X 0,Y 391.727,Z 762.261,A -85,B 0,C 180,E1 18514.214,E2 18514.214} C_VEL
LIN {X 0,Y 387.321,Z 798.196,A -85,B 0,C 180,E1 18517.435,E2 18517.435} C_VEL
LIN {X 0,Y 383.405,Z 829.181,A -85,B 0,C 180,E1 18521.278,E2 18521.278} C_VEL
LIN {X 0,Y 380.337,Z 854.563,A -85,B 0,C 180,E1 18525.588,E2 18525.588} C_VEL
LIN {X 0,Y 378.546,Z 874.17,A -85,B 0,C 180,E1 18530.211,E2 18530.211} C_VEL
LIN {X 0,Y 377.82,Z 887.684,A -85,B 0,C 180,E1 18534.827,E2 18534.827} C_VEL
LIN {X 0,Y 377.888,Z 895.164,A -85,B 0,C 180,E1 18538.854,E2 18538.854} C_VEL
LIN {X 0,Y 378.313,Z 898.679,A -85,B 0,C 180,E1 18542.298,E2 18542.298} C_VEL
LIN {X 0,Y 380.267,Z 899.089,A -85,B 0,C 180,E1 18546.867,E2 18546.867} C_VEL
LIN {X 0,Y 383.268,Z 894.777,A -85,B 0,C 180,E1 18551.401,E2 18551.401} C_VEL
LIN {X 0,Y 388.381,Z 884.412,A -85,B 0,C 180,E1 18556.291,E2 18556.291} C_VEL
LIN {X 0,Y 395.575,Z 867.952,A -85,B 0,C 180,E1 18561.043,E2 18561.043} C_VEL
LIN {X 0,Y 405.818,Z 844.001,A -85,B 0,C 180,E1 18565.721,E2 18565.721} C_VEL
LIN {X 0,Y 419.329,Z 812.705,A -85,B 0,C 180,E1 18570.086,E2 18570.086} C_VEL
LIN {X 0,Y 436.057,Z 775.559,A -85,B 0,C 180,E1 18573.772,E2 18573.772} C_VEL
LIN {X 0,Y 452.522,Z 738.129,A -85,B 0,C 180,E1 18576.309,E2 18576.309} C_VEL
LIN {X 0,Y 460.767,Z 717.596,A -85,B 0,C 180,E1 18577.303,E2 18577.303} C_VEL
LIN {X 0,Y 460.857,Z 719.542,A -85,B 0,C 180,E1 18578.185,E2 18578.185} C_VEL
LIN {X 0,Y 459.715,Z 724.438,A -85,B 0,C 180,E1 18578.669,E2 18578.669} C_VEL
LIN {X 0,Y 445.776,Z 766.498,A -85,B 0,C 180,E1 18580.684,E2 18580.684} C_VEL
LIN {X 0,Y 429.614,Z 811.005,A -85,B 0,C 180,E1 18583.862,E2 18583.862} C_VEL
LIN {X 0,Y 413.449,Z 853.576,A -85,B 0,C 180,E1 18588.208,E2 18588.208} C_VEL
LIN {X 0,Y 399.654,Z 890.222,A -85,B 0,C 180,E1 18593.343,E2 18593.343} C_VEL
LIN {X 0,Y 389.171,Z 920.394,A -85,B 0,C 180,E1 18599.024,E2 18599.024} C_VEL
LIN {X 0,Y 381.669,Z 945.188,A -85,B 0,C 180,E1 18605.243,E2 18605.243} C_VEL
LIN {X 0,Y 377.566,Z 964.523,A -85,B 0,C 180,E1 18611.886,E2 18611.886} C_VEL
LIN {X 0,Y 376.139,Z 977.397,A -85,B 0,C 180,E1 18618.387,E2 18618.387} C_VEL
LIN {X 0,Y 376.077,Z 983.161,A -85,B 0,C 180,E1 18623.064,E2 18623.064} C_VEL
LIN {X 0,Y 376.363,Z 985.934,A -85,B 0,C 180,E1 18627.699,E2 18627.699} C_VEL
LIN {X 0,Y 376.34,Z 985.615,A -85,B 0,C 180,E1 18632.314,E2 18632.314} C_VEL
LIN {X 0,Y 376.137,Z 980.846,A -85,B 0,C 180,E1 18638.112,E2 18638.112} C_VEL
LIN {X 0,Y 376.635,Z 970.876,A -85,B 0,C 180,E1 18643.975,E2 18643.975} C_VEL
LIN {X 0,Y 378.354,Z 955.812,A -85,B 0,C 180,E1 18649.772,E2 18649.772} C_VEL
LIN {X 0,Y 382.603,Z 933.607,A -85,B 0,C 180,E1 18655.832,E2 18655.832} C_VEL
LIN {X 0,Y 388.733,Z 906.552,A -85,B 0,C 180,E1 18661.268,E2 18661.268} C_VEL
LIN {X 0,Y 393.422,Z 887.17,A -85,B 0,C 180,E1 18664.338,E2 18664.338} C_VEL
LIN {X 0,Y 392.533,Z 874.996,A -85,B 0,C 180,E1 18666.18,E2 18666.18} C_VEL
LIN {X 0,Y 391.931,Z 862.274,A -85,B 0,C 180,E1 18667.947,E2 18667.947} C_VEL
LIN {X 0,Y 401.074,Z 823.414,A -85,B 0,C 180,E1 18671.937,E2 18671.937} C_VEL
LIN {X 0,Y 409.78,Z 781.221,A -85,B 0,C 180,E1 18675.071,E2 18675.071} C_VEL
LIN {X 0,Y 417.202,Z 736.502,A -85,B 0,C 180,E1 18677.368,E2 18677.368} C_VEL
LIN {X 0,Y 418.464,Z 721.142,A -85,B 0,C 180,E1 18678.018,E2 18678.018} C_VEL
LIN {X 0,Y 399.325,Z 676.143,A -85,B 0,C 180,E1 18681.245,E2 18681.245} C_VEL
LIN {X 0,Y 365.098,Z 601.31,A -85,B 0,C 180,E1 18687.014,E2 18687.014} C_VEL
LIN {X 0,Y 365.246,Z 601.31,A -85,B 0,C 180,E1 18692.852,E2 18692.852} C_VEL
LIN {X 0,Y 365.561,Z 601.31,A -85,B 0,C 180,E1 18698.099,E2 18698.099} C_VEL
LIN {X 0,Y 365.978,Z 601.31,A -85,B 0,C 180,E1 18705.617,E2 18705.617} C_VEL
LIN {X 0,Y 366.544,Z 601.31,A -85,B 0,C 180,E1 18712.875,E2 18712.875} C_VEL
LIN {X 0,Y 367.157,Z 601.31,A -85,B 0,C 180,E1 18719.997,E2 18719.997} C_VEL
LIN {X 0,Y 366.56,Z 601.31,A -85,B 0,C 180,E1 18727.173,E2 18727.173} C_VEL
LIN {X 0,Y 366.015,Z 601.31,A -85,B 0,C 180,E1 18734.376,E2 18734.376} C_VEL
LIN {X 0,Y 365.567,Z 601.31,A -85,B 0,C 180,E1 18741.895,E2 18741.895} C_VEL
LIN {X 0,Y 365.133,Z 601.31,A -85,B 0,C 180,E1 18749.855,E2 18749.855} C_VEL
LIN {X 0,Y 364.903,Z 601.476,A -85,B 0,C 180,E1 18756.266,E2 18756.266} C_VEL
LIN {X 0,Y 367.296,Z 606.974,A -85,B 0,C 180,E1 18757.131,E2 18757.131} C_VEL
LIN {X 0,Y 380.025,Z 627.625,A -85,B 0,C 180,E1 18760.855,E2 18760.855} C_VEL
LIN {X 0,Y 396.179,Z 658.385,A -85,B 0,C 180,E1 18765.172,E2 18765.172} C_VEL
LIN {X 0,Y 409.405,Z 691.082,A -85,B 0,C 180,E1 18768.732,E2 18768.732} C_VEL
LIN {X 0,Y 413.608,Z 707.158,A -85,B 0,C 180,E1 18770.324,E2 18770.324} C_VEL
LIN {X 0,Y 407.508,Z 742.84,A -85,B 0,C 180,E1 18772.653,E2 18772.653} C_VEL
LIN {X 0,Y 399.64,Z 777.975,A -85,B 0,C 180,E1 18775.908,E2 18775.908} C_VEL
LIN {X 0,Y 391.654,Z 808.178,A -85,B 0,C 180,E1 18779.799,E2 18779.799} C_VEL
LIN {X 0,Y 383.871,Z 834.952,A -85,B 0,C 180,E1 18784.527,E2 18784.527} C_VEL
LIN {X 0,Y 377.75,Z 855.151,A -85,B 0,C 180,E1 18789.446,E2 18789.446} C_VEL
LIN {X 0,Y 373.07,Z 871.931,A -85,B 0,C 180,E1 18795.288,E2 18795.288} C_VEL
LIN {X 0,Y 370.619,Z 881.729,A -85,B 0,C 180,E1 18800.581,E2 18800.581} C_VEL
LIN {X 0,Y 369.663,Z 886.639,A -85,B 0,C 180,E1 18805.291,E2 18805.291} C_VEL
LIN {X 0,Y 369.473,Z 888.31,A -85,B 0,C 180,E1 18809.994,E2 18809.994} C_VEL
LIN {X 0,Y 369.817,Z 885.66,A -85,B 0,C 180,E1 18815.873,E2 18815.873} C_VEL
LIN {X 0,Y 371.669,Z 877.294,A -85,B 0,C 180,E1 18821.996,E2 18821.996} C_VEL
LIN {X 0,Y 375.154,Z 864.185,A -85,B 0,C 180,E1 18827.598,E2 18827.598} C_VEL
LIN {X 0,Y 380.794,Z 844.931,A -85,B 0,C 180,E1 18833.13,E2 18833.13} C_VEL
LIN {X 0,Y 387.787,Z 821.384,A -85,B 0,C 180,E1 18837.954,E2 18837.954} C_VEL
LIN {X 0,Y 396.095,Z 791.632,A -85,B 0,C 180,E1 18842.374,E2 18842.374} C_VEL
LIN {X 0,Y 404.035,Z 759.229,A -85,B 0,C 180,E1 18845.855,E2 18845.855} C_VEL
LIN {X 0,Y 410.974,Z 723.196,A -85,B 0,C 180,E1 18848.635,E2 18848.635} C_VEL
LIN {X 0,Y 413.447,Z 705.544,A -85,B 0,C 180,E1 18849.7,E2 18849.7} C_VEL
LIN {X 0,Y 403.715,Z 675.412,A -85,B 0,C 180,E1 18852.775,E2 18852.775} C_VEL
LIN {X 0,Y 388.098,Z 642.136,A -85,B 0,C 180,E1 18856.823,E2 18856.823} C_VEL
LIN {X 0,Y 371.453,Z 613.405,A -85,B 0,C 180,E1 18861.479,E2 18861.479} C_VEL
LIN {X 0,Y 364.923,Z 602.304,A -85,B 0,C 180,E1 18863.532,E2 18863.532} C_VEL
LIN {X 0,Y 364.895,Z 601.31,A -85,B 0,C 180,E1 18863.968,E2 18863.968} C_VEL
LIN {X 0,Y 364.975,Z 601.31,A -85,B 0,C 180,E1 18865.019,E2 18865.019} C_VEL
LIN {X 0,Y 388.434,Z 667.626,A -85,B 0,C 180,E1 18868.988,E2 18868.988} C_VEL
LIN {X 0,Y 392.193,Z 682.55,A -85,B 0,C 180,E1 18869.718,E2 18869.718} C_VEL
LIN {X 0,Y 388.559,Z 724.714,A -85,B 0,C 180,E1 18871.436,E2 18871.436} C_VEL
LIN {X 0,Y 384.041,Z 764.295,A -85,B 0,C 180,E1 18873.974,E2 18873.974} C_VEL
LIN {X 0,Y 379.524,Z 799.782,A -85,B 0,C 180,E1 18877.255,E2 18877.255} C_VEL
LIN {X 0,Y 375.486,Z 831.274,A -85,B 0,C 180,E1 18881.288,E2 18881.288} C_VEL
LIN {X 0,Y 372.321,Z 857.297,A -85,B 0,C 180,E1 18885.873,E2 18885.873} C_VEL
LIN {X 0,Y 370.605,Z 876.451,A -85,B 0,C 180,E1 18890.593,E2 18890.593} C_VEL
LIN {X 0,Y 369.979,Z 889.604,A -85,B 0,C 180,E1 18895.306,E2 18895.306} C_VEL
LIN {X 0,Y 370.188,Z 897.523,A -85,B 0,C 180,E1 18900.003,E2 18900.003} C_VEL
LIN {X 0,Y 371.41,Z 900.64,A -85,B 0,C 180,E1 18904.682,E2 18904.682} C_VEL
LIN {X 0,Y 373.926,Z 899.028,A -85,B 0,C 180,E1 18909.329,E2 18909.329} C_VEL
LIN {X 0,Y 378.584,Z 891.55,A -85,B 0,C 180,E1 18914.486,E2 18914.486} C_VEL
LIN {X 0,Y 385.682,Z 877.245,A -85,B 0,C 180,E1 18919.715,E2 18919.715} C_VEL
LIN {X 0,Y 395.577,Z 856.385,A -85,B 0,C 180,E1 18924.615,E2 18924.615} C_VEL
LIN {X 0,Y 409.232,Z 827.294,A -85,B 0,C 180,E1 18929.375,E2 18929.375} C_VEL
LIN {X 0,Y 426.421,Z 792.388,A -85,B 0,C 180,E1 18933.414,E2 18933.414} C_VEL
LIN {X 0,Y 444.649,Z 755.911,A -85,B 0,C 180,E1 18936.351,E2 18936.351} C_VEL
LIN {X 0,Y 456.269,Z 730.717,A -85,B 0,C 180,E1 18937.765,E2 18937.765} C_VEL
LIN {X 0,Y 455.995,Z 731.959,A -85,B 0,C 180,E1 18937.967,E2 18937.967} C_VEL
LIN {X 0,Y 440.694,Z 773.253,A -85,B 0,C 180,E1 18940.089,E2 18940.089} C_VEL
LIN {X 0,Y 423.93,Z 815.198,A -85,B 0,C 180,E1 18943.269,E2 18943.269} C_VEL
LIN {X 0,Y 407.228,Z 855.866,A -85,B 0,C 180,E1 18947.601,E2 18947.601} C_VEL
LIN {X 0,Y 392.558,Z 892.224,A -85,B 0,C 180,E1 18952.916,E2 18952.916} C_VEL
LIN {X 0,Y 380.886,Z 923.79,A -85,B 0,C 180,E1 18959.198,E2 18959.198} C_VEL
LIN {X 0,Y 373.119,Z 948.98,A -85,B 0,C 180,E1 18966.048,E2 18966.048} C_VEL
LIN {X 0,Y 369.176,Z 967.863,A -85,B 0,C 180,E1 18973.31,E2 18973.31} C_VEL
LIN {X 0,Y 368.205,Z 978.228,A -85,B 0,C 180,E1 18979.335,E2 18979.335} C_VEL
LIN {X 0,Y 368.287,Z 983.98,A -85,B 0,C 180,E1 18985.287,E2 18985.287} C_VEL
LIN {X 0,Y 368.76,Z 985.18,A -85,B 0,C 180,E1 18990.006,E2 18990.006} C_VEL
LIN {X 0,Y 368.381,Z 982.204,A -85,B 0,C 180,E1 18995.909,E2 18995.909} C_VEL
LIN {X 0,Y 368.509,Z 974.162,A -85,B 0,C 180,E1 19001.87,E2 19001.87} C_VEL
LIN {X 0,Y 369.742,Z 960.721,A -85,B 0,C 180,E1 19007.906,E2 19007.906} C_VEL
LIN {X 0,Y 372.785,Z 942.448,A -85,B 0,C 180,E1 19013.671,E2 19013.671} C_VEL
LIN {X 0,Y 378.702,Z 916.147,A -85,B 0,C 180,E1 19019.686,E2 19019.686} C_VEL
LIN {X 0,Y 386.552,Z 884.217,A -85,B 0,C 180,E1 19025.05,E2 19025.05} C_VEL
LIN {X 0,Y 391.931,Z 862.274,A -85,B 0,C 180,E1 19027.947,E2 19027.947} C_VEL
LIN {X 0,Y 391.502,Z 849.14,A -85,B 0,C 180,E1 19029.65,E2 19029.65} C_VEL
LIN {X 0,Y 390.994,Z 835.36,A -85,B 0,C 180,E1 19031.25,E2 19031.25} C_VEL
LIN {X 0,Y 400.118,Z 794.426,A -85,B 0,C 180,E1 19034.671,E2 19034.671} C_VEL
LIN {X 0,Y 408.111,Z 751.074,A -85,B 0,C 180,E1 19037.23,E2 19037.23} C_VEL
LIN {X 0,Y 411.329,Z 723.443,A -85,B 0,C 180,E1 19038.473,E2 19038.473} C_VEL
LIN {X 0,Y 392.172,Z 678.032,A -85,B 0,C 180,E1 19041.823,E2 19041.823} C_VEL
LIN {X 0,Y 361.423,Z 610.849,A -85,B 0,C 180,E1 19047.182,E2 19047.182} C_VEL
LIN {X 0,Y 358.953,Z 606.365,A -85,B 0,C 180,E1 19047.941,E2 19047.941} C_VEL
LIN {X 0,Y 357.133,Z 601.31,A -85,B 0,C 180,E1 19048.782,E2 19048.782} C_VEL
LIN {X 0,Y 357.403,Z 601.31,A -85,B 0,C 180,E1 19054.918,E2 19054.918} C_VEL
LIN {X 0,Y 357.711,Z 601.31,A -85,B 0,C 180,E1 19060.193,E2 19060.193} C_VEL
LIN {X 0,Y 358.197,Z 601.31,A -85,B 0,C 180,E1 19067.789,E2 19067.789} C_VEL
LIN {X 0,Y 358.859,Z 601.31,A -85,B 0,C 180,E1 19075.154,E2 19075.154} C_VEL
LIN {X 0,Y 359.265,Z 601.31,A -85,B 0,C 180,E1 19079.997,E2 19079.997} C_VEL
LIN {X 0,Y 358.66,Z 601.31,A -85,B 0,C 180,E1 19087.277,E2 19087.277} C_VEL
LIN {X 0,Y 358.059,Z 601.31,A -85,B 0,C 180,E1 19094.702,E2 19094.702} C_VEL
LIN {X 0,Y 357.612,Z 601.31,A -85,B 0,C 180,E1 19102.408,E2 19102.408} C_VEL
LIN {X 0,Y 357.285,Z 601.31,A -85,B 0,C 180,E1 19107.797,E2 19107.797} C_VEL
LIN {X 0,Y 357.043,Z 601.888,A -85,B 0,C 180,E1 19114.393,E2 19114.393} C_VEL
LIN {X 0,Y 359.745,Z 607.247,A -85,B 0,C 180,E1 19115.402,E2 19115.402} C_VEL
LIN {X 0,Y 373.289,Z 629.229,A -85,B 0,C 180,E1 19119.651,E2 19119.651} C_VEL
LIN {X 0,Y 388.622,Z 658.006,A -85,B 0,C 180,E1 19123.971,E2 19123.971} C_VEL
LIN {X 0,Y 402.591,Z 691.443,A -85,B 0,C 180,E1 19127.839,E2 19127.839} C_VEL
LIN {X 0,Y 407.427,Z 709.227,A -85,B 0,C 180,E1 19129.686,E2 19129.686} C_VEL
LIN {X 0,Y 400.966,Z 745.483,A -85,B 0,C 180,E1 19132.108,E2 19132.108} C_VEL
LIN {X 0,Y 392.884,Z 780.043,A -85,B 0,C 180,E1 19135.387,E2 19135.387} C_VEL
LIN {X 0,Y 384.429,Z 810.808,A -85,B 0,C 180,E1 19139.457,E2 19139.457} C_VEL
LIN {X 0,Y 376.6,Z 836.542,A -85,B 0,C 180,E1 19144.136,E2 19144.136} C_VEL
LIN {X 0,Y 369.798,Z 858.154,A -85,B 0,C 180,E1 19149.611,E2 19149.611} C_VEL
LIN {X 0,Y 365.107,Z 874.224,A -85,B 0,C 180,E1 19155.575,E2 19155.575} C_VEL
LIN {X 0,Y 362.54,Z 884.233,A -85,B 0,C 180,E1 19161.582,E2 19161.582} C_VEL
LIN {X 0,Y 361.579,Z 888.874,A -85,B 0,C 180,E1 19167.592,E2 19167.592} C_VEL
LIN {X 0,Y 361.69,Z 888.823,A -85,B 0,C 180,E1 19172.394,E2 19172.394} C_VEL
LIN {X 0,Y 362.573,Z 884.12,A -85,B 0,C 180,E1 19178.404,E2 19178.404} C_VEL
LIN {X 0,Y 365.172,Z 874.023,A -85,B 0,C 180,E1 19184.409,E2 19184.409} C_VEL
LIN {X 0,Y 369.824,Z 857.847,A -85,B 0,C 180,E1 19190.374,E2 19190.374} C_VEL
LIN {X 0,Y 376.671,Z 836.02,A -85,B 0,C 180,E1 19195.872,E2 19195.872} C_VEL
LIN {X 0,Y 384.573,Z 810.03,A -85,B 0,C 180,E1 19200.554,E2 19200.554} C_VEL
LIN {X 0,Y 392.712,Z 780.613,A -85,B 0,C 180,E1 19204.432,E2 19204.432} C_VEL
LIN {X 0,Y 400.753,Z 746.197,A -85,B 0,C 180,E1 19207.729,E2 19207.729} C_VEL
LIN {X 0,Y 407.188,Z 708.245,A -85,B 0,C 180,E1 19210.302,E2 19210.302} C_VEL
LIN {X 0,Y 397.716,Z 678.326,A -85,B 0,C 180,E1 19213.468,E2 19213.468} C_VEL
LIN {X 0,Y 382.731,Z 646.221,A -85,B 0,C 180,E1 19217.523,E2 19217.523} C_VEL
LIN {X 0,Y 367.055,Z 618.987,A -85,B 0,C 180,E1 19222.089,E2 19222.089} C_VEL
LIN {X 0,Y 359.835,Z 607.337,A -85,B 0,C 180,E1 19224.423,E2 19224.423} C_VEL
LIN {X 0,Y 358.999,Z 607.593,A -85,B 0,C 180,E1 19224.741,E2 19224.741} C_VEL
LIN {X 0,Y 379.942,Z 665.392,A -85,B 0,C 180,E1 19228.33,E2 19228.33} C_VEL
LIN {X 0,Y 384.99,Z 682.29,A -85,B 0,C 180,E1 19229.237,E2 19229.237} C_VEL
LIN {X 0,Y 381.233,Z 724.983,A -85,B 0,C 180,E1 19231.01,E2 19231.01} C_VEL
LIN {X 0,Y 376.605,Z 764.288,A -85,B 0,C 180,E1 19233.581,E2 19233.581} C_VEL
LIN {X 0,Y 371.933,Z 799.958,A -85,B 0,C 180,E1 19236.923,E2 19236.923} C_VEL
LIN {X 0,Y 367.779,Z 831.611,A -85,B 0,C 180,E1 19241.03,E2 19241.03} C_VEL
LIN {X 0,Y 364.59,Z 857.202,A -85,B 0,C 180,E1 19245.567,E2 19245.567} C_VEL
LIN {X 0,Y 362.71,Z 877.686,A -85,B 0,C 180,E1 19250.689,E2 19250.689} C_VEL
LIN {X 0,Y 362.102,Z 891.432,A -85,B 0,C 180,E1 19255.805,E2 19255.805} C_VEL
LIN {X 0,Y 362.443,Z 899.71,A -85,B 0,C 180,E1 19261.2,E2 19261.2} C_VEL
LIN {X 0,Y 363.636,Z 901.855,A -85,B 0,C 180,E1 19264.782,E2 19264.782} C_VEL
LIN {X 0,Y 366.293,Z 900.596,A -85,B 0,C 180,E1 19269.525,E2 19269.525} C_VEL
LIN {X 0,Y 371.196,Z 893.525,A -85,B 0,C 180,E1 19274.781,E2 19274.781} C_VEL
LIN {X 0,Y 378.361,Z 880.555,A -85,B 0,C 180,E1 19279.9,E2 19279.9} C_VEL
LIN {X 0,Y 389.048,Z 859.941,A -85,B 0,C 180,E1 19285.056,E2 19285.056} C_VEL
LIN {X 0,Y 403.956,Z 831.172,A -85,B 0,C 180,E1 19290.024,E2 19290.024} C_VEL
LIN {X 0,Y 422.304,Z 797.586,A -85,B 0,C 180,E1 19294.093,E2 19294.093} C_VEL
LIN {X 0,Y 441.644,Z 762.487,A -85,B 0,C 180,E1 19297.046,E2 19297.046} C_VEL
LIN {X 0,Y 446.592,Z 753.099,A -85,B 0,C 180,E1 19297.634,E2 19297.634} C_VEL
LIN {X 0,Y 446.953,Z 752.87,A -85,B 0,C 180,E1 19297.893,E2 19297.893} C_VEL
LIN {X 0,Y 428.962,Z 795.458,A -85,B 0,C 180,E1 19300.594,E2 19300.594} C_VEL
LIN {X 0,Y 410.538,Z 837.164,A -85,B 0,C 180,E1 19304.461,E2 19304.461} C_VEL
LIN {X 0,Y 394.166,Z 874.159,A -85,B 0,C 180,E1 19309.203,E2 19309.203} C_VEL
LIN {X 0,Y 381.051,Z 905.296,A -85,B 0,C 180,E1 19314.564,E2 19314.564} C_VEL
LIN {X 0,Y 370.201,Z 933.858,A -85,B 0,C 180,E1 19321.172,E2 19321.172} C_VEL
LIN {X 0,Y 363.791,Z 955.453,A -85,B 0,C 180,E1 19327.992,E2 19327.992} C_VEL
LIN {X 0,Y 360.764,Z 971.807,A -85,B 0,C 180,E1 19335.411,E2 19335.411} C_VEL
LIN {X 0,Y 360.254,Z 980.55,A -85,B 0,C 180,E1 19341.929,E2 19341.929} C_VEL
LIN {X 0,Y 360.68,Z 983.986,A -85,B 0,C 180,E1 19347.599,E2 19347.599} C_VEL
LIN {X 0,Y 360.693,Z 983.488,A -85,B 0,C 180,E1 19352.414,E2 19352.414} C_VEL
LIN {X 0,Y 360.483,Z 978.779,A -85,B 0,C 180,E1 19358.145,E2 19358.145} C_VEL
LIN {X 0,Y 361.038,Z 968.051,A -85,B 0,C 180,E1 19364.591,E2 19364.591} C_VEL
LIN {X 0,Y 363.086,Z 952.077,A -85,B 0,C 180,E1 19370.739,E2 19370.739} C_VEL
LIN {X 0,Y 367.437,Z 930.692,A -85,B 0,C 180,E1 19376.652,E2 19376.652} C_VEL
LIN {X 0,Y 373.863,Z 903.93,A -85,B 0,C 180,E1 19382.144,E2 19382.144} C_VEL
LIN {X 0,Y 382.307,Z 870.86,A -85,B 0,C 180,E1 19387.194,E2 19387.194} C_VEL
LIN {X 0,Y 390.994,Z 835.36,A -85,B 0,C 180,E1 19391.25,E2 19391.25} C_VEL
LIN {X 0,Y 390.629,Z 821.244,A -85,B 0,C 180,E1 19392.774,E2 19392.774} C_VEL
LIN {X 0,Y 390.3,Z 806.708,A -85,B 0,C 180,E1 19394.217,E2 19394.217} C_VEL
LIN {X 0,Y 398.675,Z 764.683,A -85,B 0,C 180,E1 19397.046,E2 19397.046} C_VEL
LIN {X 0,Y 404.418,Z 726.087,A -85,B 0,C 180,E1 19398.895,E2 19398.895} C_VEL
LIN {X 0,Y 385.555,Z 680.991,A -85,B 0,C 180,E1 19402.323,E2 19402.323} C_VEL
LIN {X 0,Y 361.471,Z 628.022,A -85,B 0,C 180,E1 19406.585,E2 19406.585} C_VEL
LIN {X 0,Y 355.934,Z 612.885,A -85,B 0,C 180,E1 19408.466,E2 19408.466} C_VEL
LIN {X 0,Y 352.704,Z 607.851,A -85,B 0,C 180,E1 19409.496,E2 19409.496} C_VEL
LIN {X 0,Y 349.468,Z 603.254,A -85,B 0,C 180,E1 19410.562,E2 19410.562} C_VEL
LIN {X 0,Y 349.219,Z 601.31,A -85,B 0,C 180,E1 19410.908,E2 19410.908} C_VEL
LIN {X 0,Y 349.604,Z 601.31,A -85,B 0,C 180,E1 19417.043,E2 19417.043} C_VEL
LIN {X 0,Y 350.063,Z 601.31,A -85,B 0,C 180,E1 19424.948,E2 19424.948} C_VEL
LIN {X 0,Y 350.704,Z 601.31,A -85,B 0,C 180,E1 19432.551,E2 19432.551} C_VEL
LIN {X 0,Y 351.361,Z 601.31,A -85,B 0,C 180,E1 19439.997,E2 19439.997} C_VEL
LIN {X 0,Y 350.719,Z 601.31,A -85,B 0,C 180,E1 19447.442,E2 19447.442} C_VEL
LIN {X 0,Y 350.096,Z 601.31,A -85,B 0,C 180,E1 19455.044,E2 19455.044} C_VEL
LIN {X 0,Y 349.604,Z 601.31,A -85,B 0,C 180,E1 19462.95,E2 19462.95} C_VEL
LIN {X 0,Y 349.174,Z 601.31,A -85,B 0,C 180,E1 19469.773,E2 19469.773} C_VEL
LIN {X 0,Y 349.137,Z 601.794,A -85,B 0,C 180,E1 19472.3,E2 19472.3} C_VEL
LIN {X 0,Y 351.696,Z 607.132,A -85,B 0,C 180,E1 19473.349,E2 19473.349} C_VEL
LIN {X 0,Y 354.211,Z 611.089,A -85,B 0,C 180,E1 19474.278,E2 19474.278} C_VEL
LIN {X 0,Y 367.782,Z 632.427,A -85,B 0,C 180,E1 19478.722,E2 19478.722} C_VEL
LIN {X 0,Y 384.121,Z 663.931,A -85,B 0,C 180,E1 19483.554,E2 19483.554} C_VEL
LIN {X 0,Y 397.184,Z 696.385,A -85,B 0,C 180,E1 19487.397,E2 19487.397} C_VEL
LIN {X 0,Y 401.243,Z 711.389,A -85,B 0,C 180,E1 19489.029,E2 19489.029} C_VEL
LIN {X 0,Y 394.442,Z 748.13,A -85,B 0,C 180,E1 19491.543,E2 19491.543} C_VEL
LIN {X 0,Y 386.109,Z 782.362,A -85,B 0,C 180,E1 19494.882,E2 19494.882} C_VEL
LIN {X 0,Y 377.465,Z 812.614,A -85,B 0,C 180,E1 19498.976,E2 19498.976} C_VEL
LIN {X 0,Y 369.248,Z 838.394,A -85,B 0,C 180,E1 19503.788,E2 19503.788} C_VEL
LIN {X 0,Y 362.426,Z 859.163,A -85,B 0,C 180,E1 19509.177,E2 19509.177} C_VEL
LIN {X 0,Y 357.48,Z 875.23,A -85,B 0,C 180,E1 19515.26,E2 19515.26} C_VEL
LIN {X 0,Y 354.79,Z 885.226,A -85,B 0,C 180,E1 19521.397,E2 19521.397} C_VEL
LIN {X 0,Y 353.759,Z 889.861,A -85,B 0,C 180,E1 19527.538,E2 19527.538} C_VEL
LIN {X 0,Y 353.867,Z 889.81,A -85,B 0,C 180,E1 19532.447,E2 19532.447} C_VEL
LIN {X 0,Y 354.824,Z 885.111,A -85,B 0,C 180,E1 19538.589,E2 19538.589} C_VEL
LIN {X 0,Y 357.555,Z 875.031,A -85,B 0,C 180,E1 19544.723,E2 19544.723} C_VEL
LIN {X 0,Y 362.47,Z 858.854,A -85,B 0,C 180,E1 19550.806,E2 19550.806} C_VEL
LIN {X 0,Y 369.342,Z 837.895,A -85,B 0,C 180,E1 19556.215,E2 19556.215} C_VEL
LIN {X 0,Y 377.895,Z 810.779,A -85,B 0,C 180,E1 19561.203,E2 19561.203} C_VEL
LIN {X 0,Y 386.792,Z 779.712,A -85,B 0,C 180,E1 19565.315,E2 19565.315} C_VEL
LIN {X 0,Y 394.91,Z 745.48,A -85,B 0,C 180,E1 19568.563,E2 19568.563} C_VEL
LIN {X 0,Y 400.977,Z 710.897,A -85,B 0,C 180,E1 19570.927,E2 19570.927} C_VEL
LIN {X 0,Y 391.817,Z 681.477,A -85,B 0,C 180,E1 19574.159,E2 19574.159} C_VEL
LIN {X 0,Y 376.95,Z 649.416,A -85,B 0,C 180,E1 19578.371,E2 19578.371} C_VEL
LIN {X 0,Y 362.242,Z 623.711,A -85,B 0,C 180,E1 19582.862,E2 19582.862} C_VEL
LIN {X 0,Y 357.811,Z 617.768,A -85,B 0,C 180,E1 19584.257,E2 19584.257} C_VEL
LIN {X 0,Y 355.443,Z 618.676,A -85,B 0,C 180,E1 19584.841,E2 19584.841} C_VEL
LIN {X 0,Y 374.913,Z 674.367,A -85,B 0,C 180,E1 19588.286,E2 19588.286} C_VEL
LIN {X 0,Y 377.622,Z 684.735,A -85,B 0,C 180,E1 19588.836,E2 19588.836} C_VEL
LIN {X 0,Y 373.646,Z 727.244,A -85,B 0,C 180,E1 19590.691,E2 19590.691} C_VEL
LIN {X 0,Y 368.709,Z 767.879,A -85,B 0,C 180,E1 19593.464,E2 19593.464} C_VEL
LIN {X 0,Y 363.895,Z 803.854,A -85,B 0,C 180,E1 19597.002,E2 19597.002} C_VEL
LIN {X 0,Y 359.72,Z 834.468,A -85,B 0,C 180,E1 19601.156,E2 19601.156} C_VEL
LIN {X 0,Y 356.554,Z 859.801,A -85,B 0,C 180,E1 19605.863,E2 19605.863} C_VEL
LIN {X 0,Y 354.784,Z 879.381,A -85,B 0,C 180,E1 19610.938,E2 19610.938} C_VEL
LIN {X 0,Y 354.21,Z 893.251,A -85,B 0,C 180,E1 19616.325,E2 19616.325} C_VEL
LIN {X 0,Y 354.594,Z 900.589,A -85,B 0,C 180,E1 19621.227,E2 19621.227} C_VEL
LIN {X 0,Y 355.849,Z 903.026,A -85,B 0,C 180,E1 19624.887,E2 19624.887} C_VEL
LIN {X 0,Y 358.659,Z 902.109,A -85,B 0,C 180,E1 19629.73,E2 19629.73} C_VEL
LIN {X 0,Y 363.839,Z 895.552,A -85,B 0,C 180,E1 19635.087,E2 19635.087} C_VEL
LIN {X 0,Y 371.034,Z 883.75,A -85,B 0,C 180,E1 19640.092,E2 19640.092} C_VEL
LIN {X 0,Y 381.902,Z 864.823,A -85,B 0,C 180,E1 19645.244,E2 19645.244} C_VEL
LIN {X 0,Y 398.143,Z 836.375,A -85,B 0,C 180,E1 19650.509,E2 19650.509} C_VEL
LIN {X 0,Y 417.699,Z 803.868,A -85,B 0,C 180,E1 19654.68,E2 19654.68} C_VEL
LIN {X 0,Y 438.133,Z 770.357,A -85,B 0,C 180,E1 19657.647,E2 19657.647} C_VEL
LIN {X 0,Y 435.78,Z 775.685,A -85,B 0,C 180,E1 19658.134,E2 19658.134} C_VEL
LIN {X 0,Y 416.202,Z 816.833,A -85,B 0,C 180,E1 19661.343,E2 19661.343} C_VEL
LIN {X 0,Y 395.934,Z 858.986,A -85,B 0,C 180,E1 19666.09,E2 19666.09} C_VEL
LIN {X 0,Y 378.977,Z 895.131,A -85,B 0,C 180,E1 19671.798,E2 19671.798} C_VEL
LIN {X 0,Y 366.442,Z 924.76,A -85,B 0,C 180,E1 19678.213,E2 19678.213} C_VEL
LIN {X 0,Y 358.098,Z 947.921,A -85,B 0,C 180,E1 19684.975,E2 19684.975} C_VEL
LIN {X 0,Y 353.83,Z 965.092,A -85,B 0,C 180,E1 19691.92,E2 19691.92} C_VEL
LIN {X 0,Y 352.453,Z 976.488,A -85,B 0,C 180,E1 19698.852,E2 19698.852} C_VEL
LIN {X 0,Y 352.548,Z 982.101,A -85,B 0,C 180,E1 19705.076,E2 19705.076} C_VEL
LIN {X 0,Y 353.106,Z 983.131,A -85,B 0,C 180,E1 19710.007,E2 19710.007} C_VEL
LIN {X 0,Y 352.717,Z 979.796,A -85,B 0,C 180,E1 19716.172,E2 19716.172} C_VEL
LIN {X 0,Y 352.919,Z 971.455,A -85,B 0,C 180,E1 19722.403,E2 19722.403} C_VEL
LIN {X 0,Y 354.279,Z 957.421,A -85,B 0,C 180,E1 19728.716,E2 19728.716} C_VEL
LIN {X 0,Y 357.675,Z 938.671,A -85,B 0,C 180,E1 19734.658,E2 19734.658} C_VEL
LIN {X 0,Y 363.716,Z 913.416,A -85,B 0,C 180,E1 19740.542,E2 19740.542} C_VEL
LIN {X 0,Y 371.756,Z 882.304,A -85,B 0,C 180,E1 19745.912,E2 19745.912} C_VEL
LIN {X 0,Y 380.909,Z 846.707,A -85,B 0,C 180,E1 19750.463,E2 19750.463} C_VEL
LIN {X 0,Y 390.136,Z 807.478,A -85,B 0,C 180,E1 19754.157,E2 19754.157} C_VEL
LIN {X 0,Y 390.3,Z 806.708,A -85,B 0,C 180,E1 19754.217,E2 19754.217} C_VEL
LIN {X 0,Y 389.785,Z 791.87,A -85,B 0,C 180,E1 19755.581,E2 19755.581} C_VEL
LIN {X 0,Y 389.017,Z 778.572,A -85,B 0,C 180,E1 19756.722,E2 19756.722} C_VEL
LIN {X 0,Y 389.353,Z 776.556,A -85,B 0,C 180,E1 19756.852,E2 19756.852} C_VEL
LIN {X 0,Y 396.608,Z 734.909,A -85,B 0,C 180,E1 19759.047,E2 19759.047} C_VEL
LIN {X 0,Y 397.093,Z 727.837,A -85,B 0,C 180,E1 19759.385,E2 19759.385} C_VEL
LIN {X 0,Y 379.817,Z 686.053,A -85,B 0,C 180,E1 19762.669,E2 19762.669} C_VEL
LIN {X 0,Y 361.168,Z 644.263,A -85,B 0,C 180,E1 19766.053,E2 19766.053} C_VEL
LIN {X 0,Y 352.703,Z 619.092,A -85,B 0,C 180,E1 19769.077,E2 19769.077} C_VEL
LIN {X 0,Y 344.895,Z 607.893,A -85,B 0,C 180,E1 19771.706,E2 19771.706} C_VEL
LIN {X 0,Y 341.616,Z 603.275,A -85,B 0,C 180,E1 19772.912,E2 19772.912} C_VEL
LIN {X 0,Y 341.383,Z 601.31,A -85,B 0,C 180,E1 19773.185,E2 19773.185} C_VEL
LIN {X 0,Y 341.781,Z 601.31,A -85,B 0,C 180,E1 19779.229,E2 19779.229} C_VEL
LIN {X 0,Y 342.312,Z 601.31,A -85,B 0,C 180,E1 19787.213,E2 19787.213} C_VEL
LIN {X 0,Y 343.018,Z 601.31,A -85,B 0,C 180,E1 19794.929,E2 19794.929} C_VEL
LIN {X 0,Y 343.47,Z 601.31,A -85,B 0,C 180,E1 19799.997,E2 19799.997} C_VEL
LIN {X 0,Y 342.776,Z 601.31,A -85,B 0,C 180,E1 19807.616,E2 19807.616} C_VEL
LIN {X 0,Y 342.152,Z 601.31,A -85,B 0,C 180,E1 19815.402,E2 19815.402} C_VEL
LIN {X 0,Y 341.656,Z 601.31,A -85,B 0,C 180,E1 19823.516,E2 19823.516} C_VEL
LIN {X 0,Y 341.286,Z 601.587,A -85,B 0,C 180,E1 19829.958,E2 19829.958} C_VEL
LIN {X 0,Y 343.54,Z 606.888,A -85,B 0,C 180,E1 19831.023,E2 19831.023} C_VEL
LIN {X 0,Y 346.026,Z 610.026,A -85,B 0,C 180,E1 19831.976,E2 19831.976} C_VEL
LIN {X 0,Y 360.797,Z 633.372,A -85,B 0,C 180,E1 19837.281,E2 19837.281} C_VEL
LIN {X 0,Y 376.603,Z 663.426,A -85,B 0,C 180,E1 19842.245,E2 19842.245} C_VEL
LIN {X 0,Y 389.729,Z 694.912,A -85,B 0,C 180,E1 19846.215,E2 19846.215} C_VEL
LIN {X 0,Y 394.979,Z 714.672,A -85,B 0,C 180,E1 19848.425,E2 19848.425} C_VEL
LIN {X 0,Y 387.969,Z 750.774,A -85,B 0,C 180,E1 19850.96,E2 19850.96} C_VEL
LIN {X 0,Y 379.244,Z 785.15,A -85,B 0,C 180,E1 19854.414,E2 19854.414} C_VEL
LIN {X 0,Y 370.304,Z 815.067,A -85,B 0,C 180,E1 19858.576,E2 19858.576} C_VEL
LIN {X 0,Y 361.688,Z 840.852,A -85,B 0,C 180,E1 19863.562,E2 19863.562} C_VEL
LIN {X 0,Y 354.421,Z 862.123,A -85,B 0,C 180,E1 19869.34,E2 19869.34} C_VEL
LIN {X 0,Y 349.494,Z 877.47,A -85,B 0,C 180,E1 19875.558,E2 19875.558} C_VEL
LIN {X 0,Y 347.035,Z 886.219,A -85,B 0,C 180,E1 19881.203,E2 19881.203} C_VEL
LIN {X 0,Y 345.95,Z 890.846,A -85,B 0,C 180,E1 19887.483,E2 19887.483} C_VEL
LIN {X 0,Y 346.043,Z 890.798,A -85,B 0,C 180,E1 19892.503,E2 19892.503} C_VEL
LIN {X 0,Y 347.068,Z 886.107,A -85,B 0,C 180,E1 19898.782,E2 19898.782} C_VEL
LIN {X 0,Y 349.959,Z 876.037,A -85,B 0,C 180,E1 19905.05,E2 19905.05} C_VEL
LIN {X 0,Y 355.108,Z 859.872,A -85,B 0,C 180,E1 19911.258,E2 19911.258} C_VEL
LIN {X 0,Y 362.233,Z 839.137,A -85,B 0,C 180,E1 19916.715,E2 19916.715} C_VEL
LIN {X 0,Y 371.046,Z 812.359,A -85,B 0,C 180,E1 19921.744,E2 19921.744} C_VEL
LIN {X 0,Y 380.047,Z 782.11,A -85,B 0,C 180,E1 19925.836,E2 19925.836} C_VEL
LIN {X 0,Y 388.468,Z 748.115,A -85,B 0,C 180,E1 19929.145,E2 19929.145} C_VEL
LIN {X 0,Y 394.74,Z 713.09,A -85,B 0,C 180,E1 19931.614,E2 19931.614} C_VEL
LIN {X 0,Y 386.023,Z 684.804,A -85,B 0,C 180,E1 19934.852,E2 19934.852} C_VEL
LIN {X 0,Y 371.568,Z 653.187,A -85,B 0,C 180,E1 19939.152,E2 19939.152} C_VEL
LIN {X 0,Y 356.811,Z 626.925,A -85,B 0,C 180,E1 19943.913,E2 19943.913} C_VEL
LIN {X 0,Y 352.371,Z 629.848,A -85,B 0,C 180,E1 19944.799,E2 19944.799} C_VEL
LIN {X 0,Y 352.627,Z 631.915,A -85,B 0,C 180,E1 19945.099,E2 19945.099} C_VEL
LIN {X 0,Y 370.244,Z 684.656,A -85,B 0,C 180,E1 19948.338,E2 19948.338} C_VEL
LIN {X 0,Y 366.298,Z 727.466,A -85,B 0,C 180,E1 19950.249,E2 19950.249} C_VEL
LIN {X 0,Y 361.28,Z 767.807,A -85,B 0,C 180,E1 19953.043,E2 19953.043} C_VEL
LIN {X 0,Y 356.358,Z 803.547,A -85,B 0,C 180,E1 19956.597,E2 19956.597} C_VEL
LIN {X 0,Y 352.083,Z 834.234,A -85,B 0,C 180,E1 19960.811,E2 19960.811} C_VEL
LIN {X 0,Y 348.846,Z 859.594,A -85,B 0,C 180,E1 19965.544,E2 19965.544} C_VEL
LIN {X 0,Y 347.001,Z 879.068,A -85,B 0,C 180,E1 19970.581,E2 19970.581} C_VEL
LIN {X 0,Y 346.404,Z 892.549,A -85,B 0,C 180,E1 19975.614,E2 19975.614} C_VEL
LIN {X 0,Y 346.627,Z 900.011,A -85,B 0,C 180,E1 19980.003,E2 19980.003} C_VEL
LIN {X 0,Y 348.066,Z 904.145,A -85,B 0,C 180,E1 19984.997,E2 19984.997} C_VEL
LIN {X 0,Y 351.039,Z 903.608,A -85,B 0,C 180,E1 19989.943,E2 19989.943} C_VEL
LIN {X 0,Y 355.743,Z 898.517,A -85,B 0,C 180,E1 19994.806,E2 19994.806} C_VEL
LIN {X 0,Y 364.051,Z 886.424,A -85,B 0,C 180,E1 20000.494,E2 20000.494} C_VEL
LIN {X 0,Y 376.14,Z 867.289,A -85,B 0,C 180,E1 20005.979,E2 20005.979} C_VEL
LIN {X 0,Y 393.587,Z 839.639,A -85,B 0,C 180,E1 20011.309,E2 20011.309} C_VEL
LIN {X 0,Y 414.363,Z 808.31,A -85,B 0,C 180,E1 20015.48,E2 20015.48} C_VEL
LIN {X 0,Y 429.021,Z 786.591,A -85,B 0,C 180,E1 20017.591,E2 20017.591} C_VEL
LIN {X 0,Y 428.97,Z 787.013,A -85,B 0,C 180,E1 20017.801,E2 20017.801} C_VEL
LIN {X 0,Y 408.961,Z 825.317,A -85,B 0,C 180,E1 20021.084,E2 20021.084} C_VEL
LIN {X 0,Y 388.677,Z 864.136,A -85,B 0,C 180,E1 20025.788,E2 20025.788} C_VEL
LIN {X 0,Y 370.746,Z 900.035,A -85,B 0,C 180,E1 20031.868,E2 20031.868} C_VEL
LIN {X 0,Y 357.357,Z 929.784,A -85,B 0,C 180,E1 20038.859,E2 20038.859} C_VEL
LIN {X 0,Y 349.18,Z 952.381,A -85,B 0,C 180,E1 20046.212,E2 20046.212} C_VEL
LIN {X 0,Y 345.28,Z 969.166,A -85,B 0,C 180,E1 20054.089,E2 20054.089} C_VEL
LIN {X 0,Y 344.528,Z 978.429,A -85,B 0,C 180,E1 20061.225,E2 20061.225} C_VEL
LIN {X 0,Y 345.004,Z 981.993,A -85,B 0,C 180,E1 20067.49,E2 20067.49} C_VEL
LIN {X 0,Y 345.032,Z 981.297,A -85,B 0,C 180,E1 20072.524,E2 20072.524} C_VEL
LIN {X 0,Y 344.858,Z 977.34,A -85,B 0,C 180,E1 20077.581,E2 20077.581} C_VEL
LIN {X 0,Y 345.271,Z 967.558,A -85,B 0,C 180,E1 20083.974,E2 20083.974} C_VEL
LIN {X 0,Y 347.136,Z 952.099,A -85,B 0,C 180,E1 20090.445,E2 20090.445} C_VEL
LIN {X 0,Y 351.758,Z 930.178,A -85,B 0,C 180,E1 20096.898,E2 20096.898} C_VEL
LIN {X 0,Y 358.237,Z 904.083,A -85,B 0,C 180,E1 20102.54,E2 20102.54} C_VEL
LIN {X 0,Y 367.172,Z 870.743,A -85,B 0,C 180,E1 20107.876,E2 20107.876} C_VEL
LIN {X 0,Y 376.675,Z 833.532,A -85,B 0,C 180,E1 20112.265,E2 20112.265} C_VEL
LIN {X 0,Y 386.089,Z 792.803,A -85,B 0,C 180,E1 20115.752,E2 20115.752} C_VEL
LIN {X 0,Y 389.353,Z 776.556,A -85,B 0,C 180,E1 20116.852,E2 20116.852} C_VEL
LIN {X 0,Y 389.537,Z 764.789,A -85,B 0,C 180,E1 20117.716,E2 20117.716} C_VEL
LIN {X 0,Y 387.928,Z 747.112,A -85,B 0,C 180,E1 20119.02,E2 20119.02} C_VEL
LIN {X 0,Y 388.182,Z 745.058,A -85,B 0,C 180,E1 20119.126,E2 20119.126} C_VEL
LIN {X 0,Y 389.933,Z 729.948,A -85,B 0,C 180,E1 20119.856,E2 20119.856} C_VEL
LIN {X 0,Y 372.411,Z 687.286,A -85,B 0,C 180,E1 20123.309,E2 20123.309} C_VEL
LIN {X 0,Y 360.062,Z 659.019,A -85,B 0,C 180,E1 20125.661,E2 20125.661} C_VEL
LIN {X 0,Y 349.219,Z 624.877,A -85,B 0,C 180,E1 20129.769,E2 20129.769} C_VEL
LIN {X 0,Y 341.372,Z 614.053,A -85,B 0,C 180,E1 20132.522,E2 20132.522} C_VEL
LIN {X 0,Y 337.244,Z 608.019,A -85,B 0,C 180,E1 20134.137,E2 20134.137} C_VEL
LIN {X 0,Y 333.842,Z 603.266,A -85,B 0,C 180,E1 20135.559,E2 20135.559} C_VEL
LIN {X 0,Y 333.634,Z 601.31,A -85,B 0,C 180,E1 20135.876,E2 20135.876} C_VEL
LIN {X 0,Y 334.049,Z 601.31,A -85,B 0,C 180,E1 20142.299,E2 20142.299} C_VEL
LIN {X 0,Y 334.545,Z 601.31,A -85,B 0,C 180,E1 20149.561,E2 20149.561} C_VEL
LIN {X 0,Y 335.28,Z 601.31,A -85,B 0,C 180,E1 20157.407,E2 20157.407} C_VEL
LIN {X 0,Y 335.318,Z 601.31,A -85,B 0,C 180,E1 20162.586,E2 20162.586} C_VEL
LIN {X 0,Y 334.57,Z 601.31,A -85,B 0,C 180,E1 20170.431,E2 20170.431} C_VEL
LIN {X 0,Y 334.004,Z 601.31,A -85,B 0,C 180,E1 20178.508,E2 20178.508} C_VEL
LIN {X 0,Y 333.584,Z 601.31,A -85,B 0,C 180,E1 20184.692,E2 20184.692} C_VEL
LIN {X 0,Y 333.483,Z 602.004,A -85,B 0,C 180,E1 20187.35,E2 20187.35} C_VEL
LIN {X 0,Y 336.043,Z 607.22,A -85,B 0,C 180,E1 20188.671,E2 20188.671} C_VEL
LIN {X 0,Y 338.309,Z 609.995,A -85,B 0,C 180,E1 20189.625,E2 20189.625} C_VEL
LIN {X 0,Y 350.62,Z 629.366,A -85,B 0,C 180,E1 20194.58,E2 20194.58} C_VEL
LIN {X 0,Y 364.676,Z 653.911,A -85,B 0,C 180,E1 20199.401,E2 20199.401} C_VEL
LIN {X 0,Y 379.098,Z 685.039,A -85,B 0,C 180,E1 20203.918,E2 20203.918} C_VEL
LIN {X 0,Y 388.385,Z 713.934,A -85,B 0,C 180,E1 20207.406,E2 20207.406} C_VEL
LIN {X 0,Y 388.448,Z 719.718,A -85,B 0,C 180,E1 20207.907,E2 20207.907} C_VEL
LIN {X 0,Y 380.915,Z 756.167,A -85,B 0,C 180,E1 20210.614,E2 20210.614} C_VEL
LIN {X 0,Y 371.987,Z 789.449,A -85,B 0,C 180,E1 20214.114,E2 20214.114} C_VEL
LIN {X 0,Y 362.527,Z 819.337,A -85,B 0,C 180,E1 20218.496,E2 20218.496} C_VEL
LIN {X 0,Y 353.534,Z 845.017,A -85,B 0,C 180,E1 20223.724,E2 20223.724} C_VEL
LIN {X 0,Y 346.379,Z 864.923,A -85,B 0,C 180,E1 20229.508,E2 20229.508} C_VEL
LIN {X 0,Y 341.481,Z 879.709,A -85,B 0,C 180,E1 20235.867,E2 20235.867} C_VEL
LIN {X 0,Y 338.863,Z 888.591,A -85,B 0,C 180,E1 20242.284,E2 20242.284} C_VEL
LIN {X 0,Y 338.129,Z 891.834,A -85,B 0,C 180,E1 20247.425,E2 20247.425} C_VEL
LIN {X 0,Y 338.221,Z 891.786,A -85,B 0,C 180,E1 20252.561,E2 20252.561} C_VEL
LIN {X 0,Y 339.297,Z 887.105,A -85,B 0,C 180,E1 20258.985,E2 20258.985} C_VEL
LIN {X 0,Y 342.357,Z 877.049,A -85,B 0,C 180,E1 20265.392,E2 20265.392} C_VEL
LIN {X 0,Y 347.778,Z 860.89,A -85,B 0,C 180,E1 20271.728,E2 20271.728} C_VEL
LIN {X 0,Y 355.21,Z 840.179,A -85,B 0,C 180,E1 20277.286,E2 20277.286} C_VEL
LIN {X 0,Y 364.343,Z 813.548,A -85,B 0,C 180,E1 20282.366,E2 20282.366} C_VEL
LIN {X 0,Y 373.709,Z 783.15,A -85,B 0,C 180,E1 20286.54,E2 20286.54} C_VEL
LIN {X 0,Y 382.412,Z 749.107,A -85,B 0,C 180,E1 20289.887,E2 20289.887} C_VEL
LIN {X 0,Y 388.712,Z 716.151,A -85,B 0,C 180,E1 20292.233,E2 20292.233} C_VEL
LIN {X 0,Y 380.348,Z 688.217,A -85,B 0,C 180,E1 20295.546,E2 20295.546} C_VEL
LIN {X 0,Y 366.47,Z 657.671,A -85,B 0,C 180,E1 20299.868,E2 20299.868} C_VEL
LIN {X 0,Y 354.963,Z 636.796,A -85,B 0,C 180,E1 20303.695,E2 20303.695} C_VEL
LIN {X 0,Y 352.908,Z 637.853,A -85,B 0,C 180,E1 20304.117,E2 20304.117} C_VEL
LIN {X 0,Y 349.365,Z 641.379,A -85,B 0,C 180,E1 20304.747,E2 20304.747} C_VEL
LIN {X 0,Y 348.324,Z 641.925,A -85,B 0,C 180,E1 20305.13,E2 20305.13} C_VEL
LIN {X 0,Y 362.99,Z 687.214,A -85,B 0,C 180,E1 20307.93,E2 20307.93} C_VEL
LIN {X 0,Y 358.706,Z 730.006,A -85,B 0,C 180,E1 20309.922,E2 20309.922} C_VEL
LIN {X 0,Y 353.635,Z 769.478,A -85,B 0,C 180,E1 20312.757,E2 20312.757} C_VEL
LIN {X 0,Y 348.432,Z 806.313,A -85,B 0,C 180,E1 20316.562,E2 20316.562} C_VEL
LIN {X 0,Y 343.973,Z 837.418,A -85,B 0,C 180,E1 20321.012,E2 20321.012} C_VEL
LIN {X 0,Y 340.787,Z 862.18,A -85,B 0,C 180,E1 20325.852,E2 20325.852} C_VEL
LIN {X 0,Y 339.025,Z 881.26,A -85,B 0,C 180,E1 20331.006,E2 20331.006} C_VEL
LIN {X 0,Y 338.509,Z 894.342,A -85,B 0,C 180,E1 20336.154,E2 20336.154} C_VEL
LIN {X 0,Y 338.917,Z 902.357,A -85,B 0,C 180,E1 20341.284,E2 20341.284} C_VEL
LIN {X 0,Y 340.276,Z 905.261,A -85,B 0,C 180,E1 20345.112,E2 20345.112} C_VEL
LIN {X 0,Y 343.415,Z 905.103,A -85,B 0,C 180,E1 20350.166,E2 20350.166} C_VEL
LIN {X 0,Y 348.36,Z 900.469,A -85,B 0,C 180,E1 20355.128,E2 20355.128} C_VEL
LIN {X 0,Y 356.732,Z 889.612,A -85,B 0,C 180,E1 20360.711,E2 20360.711} C_VEL
LIN {X 0,Y 368.988,Z 871.969,A -85,B 0,C 180,E1 20366.193,E2 20366.193} C_VEL
LIN {X 0,Y 387.87,Z 844.809,A -85,B 0,C 180,E1 20371.824,E2 20371.824} C_VEL
LIN {X 0,Y 410.601,Z 813.799,A -85,B 0,C 180,E1 20376.182,E2 20376.182} C_VEL
LIN {X 0,Y 419.889,Z 801.216,A -85,B 0,C 180,E1 20377.507,E2 20377.507} C_VEL
LIN {X 0,Y 417.944,Z 805.067,A -85,B 0,C 180,E1 20378.041,E2 20378.041} C_VEL
LIN {X 0,Y 395.678,Z 844.016,A -85,B 0,C 180,E1 20382.039,E2 20382.039} C_VEL
LIN {X 0,Y 375.769,Z 879.501,A -85,B 0,C 180,E1 20387.13,E2 20387.13} C_VEL
LIN {X 0,Y 359.221,Z 911.054,A -85,B 0,C 180,E1 20393.372,E2 20393.372} C_VEL
LIN {X 0,Y 347.043,Z 937.521,A -85,B 0,C 180,E1 20400.54,E2 20400.54} C_VEL
LIN {X 0,Y 339.736,Z 958.302,A -85,B 0,C 180,E1 20408.419,E2 20408.419} C_VEL
LIN {X 0,Y 337.001,Z 971.756,A -85,B 0,C 180,E1 20415.928,E2 20415.928} C_VEL
LIN {X 0,Y 336.716,Z 978.534,A -85,B 0,C 180,E1 20422.249,E2 20422.249} C_VEL
LIN {X 0,Y 337.162,Z 980.923,A -85,B 0,C 180,E1 20427.431,E2 20427.431} C_VEL
LIN {X 0,Y 337.2,Z 980.116,A -85,B 0,C 180,E1 20432.583,E2 20432.583} C_VEL
LIN {X 0,Y 336.979,Z 975.118,A -85,B 0,C 180,E1 20438.483,E2 20438.483} C_VEL
LIN {X 0,Y 337.539,Z 964.901,A -85,B 0,C 180,E1 20444.904,E2 20444.904} C_VEL
LIN {X 0,Y 340.297,Z 946.573,A -85,B 0,C 180,E1 20452.247,E2 20452.247} C_VEL
LIN {X 0,Y 345.198,Z 924.946,A -85,B 0,C 180,E1 20458.412,E2 20458.412} C_VEL
LIN {X 0,Y 352.095,Z 898.179,A -85,B 0,C 180,E1 20463.833,E2 20463.833} C_VEL
LIN {X 0,Y 360.802,Z 865.955,A -85,B 0,C 180,E1 20468.86,E2 20468.86} C_VEL
LIN {X 0,Y 370.25,Z 829.783,A -85,B 0,C 180,E1 20473.063,E2 20473.063} C_VEL
LIN {X 0,Y 379.504,Z 790.221,A -85,B 0,C 180,E1 20476.432,E2 20476.432} C_VEL
LIN {X 0,Y 387.756,Z 747.715,A -85,B 0,C 180,E1 20478.995,E2 20478.995} C_VEL
LIN {X 0,Y 388.182,Z 745.058,A -85,B 0,C 180,E1 20479.126,E2 20479.126} C_VEL
LIN {X 0,Y 386.951,Z 737.387,A -85,B 0,C 180,E1 20479.689,E2 20479.689} C_VEL
LIN {X 0,Y 380.5,Z 725.899,A -85,B 0,C 180,E1 20480.863,E2 20480.863} C_VEL
LIN {X 0,Y 361.066,Z 679.578,A -85,B 0,C 180,E1 20484.672,E2 20484.672} C_VEL
LIN {X 0,Y 345.783,Z 630.638,A -85,B 0,C 180,E1 20490.467,E2 20490.467} C_VEL
LIN {X 0,Y 334.311,Z 614.719,A -85,B 0,C 180,E1 20494.805,E2 20494.805} C_VEL
LIN {X 0,Y 329.788,Z 608.218,A -85,B 0,C 180,E1 20496.818,E2 20496.818} C_VEL
LIN {X 0,Y 326.32,Z 603.769,A -85,B 0,C 180,E1 20498.484,E2 20498.484} C_VEL
LIN {X 0,Y 325.98,Z 601.31,A -85,B 0,C 180,E1 20498.818,E2 20498.818} C_VEL
LIN {X 0,Y 326.479,Z 601.31,A -85,B 0,C 180,E1 20507.096,E2 20507.096} C_VEL
LIN {X 0,Y 327.176,Z 601.31,A -85,B 0,C 180,E1 20514.683,E2 20514.683} C_VEL
LIN {X 0,Y 327.659,Z 601.31,A -85,B 0,C 180,E1 20519.997,E2 20519.997} C_VEL
LIN {X 0,Y 326.89,Z 601.31,A -85,B 0,C 180,E1 20527.988,E2 20527.988} C_VEL
LIN {X 0,Y 326.48,Z 601.31,A -85,B 0,C 180,E1 20533.412,E2 20533.412} C_VEL
LIN {X 0,Y 325.86,Z 601.31,A -85,B 0,C 180,E1 20541.83,E2 20541.83} C_VEL
LIN {X 0,Y 325.74,Z 601.902,A -85,B 0,C 180,E1 20544.282,E2 20544.282} C_VEL
LIN {X 0,Y 328.271,Z 607.257,A -85,B 0,C 180,E1 20545.833,E2 20545.833} C_VEL
LIN {X 0,Y 330.667,Z 610.011,A -85,B 0,C 180,E1 20546.986,E2 20546.986} C_VEL
LIN {X 0,Y 340.084,Z 624.674,A -85,B 0,C 180,E1 20551.319,E2 20551.319} C_VEL
LIN {X 0,Y 353.572,Z 646.826,A -85,B 0,C 180,E1 20556.502,E2 20556.502} C_VEL
LIN {X 0,Y 367.947,Z 675.601,A -85,B 0,C 180,E1 20561.396,E2 20561.396} C_VEL
LIN {X 0,Y 379.176,Z 704.814,A -85,B 0,C 180,E1 20565.258,E2 20565.258} C_VEL
LIN {X 0,Y 382.607,Z 720.879,A -85,B 0,C 180,E1 20567.136,E2 20567.136} C_VEL
LIN {X 0,Y 374.823,Z 757.484,A -85,B 0,C 180,E1 20569.884,E2 20569.884} C_VEL
LIN {X 0,Y 365.594,Z 790.712,A -85,B 0,C 180,E1 20573.424,E2 20573.424} C_VEL
LIN {X 0,Y 355.841,Z 820.384,A -85,B 0,C 180,E1 20577.835,E2 20577.835} C_VEL
LIN {X 0,Y 346.683,Z 845.515,A -85,B 0,C 180,E1 20583.027,E2 20583.027} C_VEL
LIN {X 0,Y 339.028,Z 865.928,A -85,B 0,C 180,E1 20589.043,E2 20589.043} C_VEL
LIN {X 0,Y 333.871,Z 880.707,A -85,B 0,C 180,E1 20595.538,E2 20595.538} C_VEL
LIN {X 0,Y 331.081,Z 889.587,A -85,B 0,C 180,E1 20602.101,E2 20602.101} C_VEL
LIN {X 0,Y 330.305,Z 892.821,A -85,B 0,C 180,E1 20607.364,E2 20607.364} C_VEL
LIN {X 0,Y 330.409,Z 892.772,A -85,B 0,C 180,E1 20612.621,E2 20612.621} C_VEL
LIN {X 0,Y 331.537,Z 888.1,A -85,B 0,C 180,E1 20619.197,E2 20619.197} C_VEL
LIN {X 0,Y 334.774,Z 878.06,A -85,B 0,C 180,E1 20625.75,E2 20625.75} C_VEL
LIN {X 0,Y 340.482,Z 861.917,A -85,B 0,C 180,E1 20632.219,E2 20632.219} C_VEL
LIN {X 0,Y 348.244,Z 841.213,A -85,B 0,C 180,E1 20637.879,E2 20637.879} C_VEL
LIN {X 0,Y 357.717,Z 814.572,A -85,B 0,C 180,E1 20643.041,E2 20643.041} C_VEL
LIN {X 0,Y 367.45,Z 784.183,A -85,B 0,C 180,E1 20647.267,E2 20647.267} C_VEL
LIN {X 0,Y 376.397,Z 750.291,A -85,B 0,C 180,E1 20650.638,E2 20650.638} C_VEL
LIN {X 0,Y 382.717,Z 719.22,A -85,B 0,C 180,E1 20652.871,E2 20652.871} C_VEL
LIN {X 0,Y 374.633,Z 691.435,A -85,B 0,C 180,E1 20656.295,E2 20656.295} C_VEL
LIN {X 0,Y 360.511,Z 660.022,A -85,B 0,C 180,E1 20660.931,E2 20660.931} C_VEL
LIN {X 0,Y 352.647,Z 646.242,A -85,B 0,C 180,E1 20663.609,E2 20663.609} C_VEL
LIN {X 0,Y 345.467,Z 652.851,A -85,B 0,C 180,E1 20664.897,E2 20664.897} C_VEL
LIN {X 0,Y 344.485,Z 653.277,A -85,B 0,C 180,E1 20665.25,E2 20665.25} C_VEL
LIN {X 0,Y 355.736,Z 688.427,A -85,B 0,C 180,E1 20667.455,E2 20667.455} C_VEL
LIN {X 0,Y 351.178,Z 731.619,A -85,B 0,C 180,E1 20669.544,E2 20669.544} C_VEL
LIN {X 0,Y 345.712,Z 772.561,A -85,B 0,C 180,E1 20672.61,E2 20672.61} C_VEL
LIN {X 0,Y 340.409,Z 809.299,A -85,B 0,C 180,E1 20676.567,E2 20676.567} C_VEL
LIN {X 0,Y 336.011,Z 839.585,A -85,B 0,C 180,E1 20681.055,E2 20681.055} C_VEL
LIN {X 0,Y 332.761,Z 864.692,A -85,B 0,C 180,E1 20686.176,E2 20686.176} C_VEL
LIN {X 0,Y 331.07,Z 883.357,A -85,B 0,C 180,E1 20691.451,E2 20691.451} C_VEL
LIN {X 0,Y 330.664,Z 896.1,A -85,B 0,C 180,E1 20696.72,E2 20696.72} C_VEL
LIN {X 0,Y 331.405,Z 904.579,A -85,B 0,C 180,E1 20702.623,E2 20702.623} C_VEL
LIN {X 0,Y 334.02,Z 907.063,A -85,B 0,C 180,E1 20707.823,E2 20707.823} C_VEL
LIN {X 0,Y 338.134,Z 905.078,A -85,B 0,C 180,E1 20712.948,E2 20712.948} C_VEL
LIN {X 0,Y 345.319,Z 897.719,A -85,B 0,C 180,E1 20718.548,E2 20718.548} C_VEL
LIN {X 0,Y 356.785,Z 883.18,A -85,B 0,C 180,E1 20724.458,E2 20724.458} C_VEL
LIN {X 0,Y 373.501,Z 861.241,A -85,B 0,C 180,E1 20730.13,E2 20730.13} C_VEL
LIN {X 0,Y 394.381,Z 834.712,A -85,B 0,C 180,E1 20734.849,E2 20734.849} C_VEL
LIN {X 0,Y 411.338,Z 813.785,A -85,B 0,C 180,E1 20737.521,E2 20737.521} C_VEL
LIN {X 0,Y 382.861,Z 859.711,A -85,B 0,C 180,E1 20742.942,E2 20742.942} C_VEL
LIN {X 0,Y 362.178,Z 894.514,A -85,B 0,C 180,E1 20748.845,E2 20748.845} C_VEL
LIN {X 0,Y 345.795,Z 924.995,A -85,B 0,C 180,E1 20756.083,E2 20756.083} C_VEL
LIN {X 0,Y 334.954,Z 949.308,A -85,B 0,C 180,E1 20764.196,E2 20764.196} C_VEL
LIN {X 0,Y 329.89,Z 966.591,A -85,B 0,C 180,E1 20772.637,E2 20772.637} C_VEL
LIN {X 0,Y 328.786,Z 975.31,A -85,B 0,C 180,E1 20779.385,E2 20779.385} C_VEL
LIN {X 0,Y 328.998,Z 979.082,A -85,B 0,C 180,E1 20784.722,E2 20784.722} C_VEL
LIN {X 0,Y 329.635,Z 979.822,A -85,B 0,C 180,E1 20790.007,E2 20790.007} C_VEL
LIN {X 0,Y 329.251,Z 976.024,A -85,B 0,C 180,E1 20796.614,E2 20796.614} C_VEL
LIN {X 0,Y 329.512,Z 966.914,A -85,B 0,C 180,E1 20803.3,E2 20803.3} C_VEL
LIN {X 0,Y 331.866,Z 949.215,A -85,B 0,C 180,E1 20811.431,E2 20811.431} C_VEL
LIN {X 0,Y 336.577,Z 929.02,A -85,B 0,C 180,E1 20817.747,E2 20817.747} C_VEL
LIN {X 0,Y 343.031,Z 904.699,A -85,B 0,C 180,E1 20823.187,E2 20823.187} C_VEL
LIN {X 0,Y 350.749,Z 875.484,A -85,B 0,C 180,E1 20827.922,E2 20827.922} C_VEL
LIN {X 0,Y 361.847,Z 833.77,A -85,B 0,C 180,E1 20833.1,E2 20833.1} C_VEL
LIN {X 0,Y 371.785,Z 792.723,A -85,B 0,C 180,E1 20836.753,E2 20836.753} C_VEL
LIN {X 0,Y 380.343,Z 750.279,A -85,B 0,C 180,E1 20839.415,E2 20839.415} C_VEL
LIN {X 0,Y 382.76,Z 731.985,A -85,B 0,C 180,E1 20840.33,E2 20840.33} C_VEL
LIN {X 0,Y 380.5,Z 725.899,A -85,B 0,C 180,E1 20840.863,E2 20840.863} C_VEL
LIN {X 0,Y 371.666,Z 713.824,A -85,B 0,C 180,E1 20842.258,E2 20842.258} C_VEL
LIN {X 0,Y 362.669,Z 701.584,A -85,B 0,C 180,E1 20843.634,E2 20843.634} C_VEL
LIN {X 0,Y 356.128,Z 684.956,A -85,B 0,C 180,E1 20845.195,E2 20845.195} C_VEL
LIN {X 0,Y 342.256,Z 636.169,A -85,B 0,C 180,E1 20851.223,E2 20851.223} C_VEL
LIN {X 0,Y 331.334,Z 621.214,A -85,B 0,C 180,E1 20855.518,E2 20855.518} C_VEL
LIN {X 0,Y 326.97,Z 615.051,A -85,B 0,C 180,E1 20857.535,E2 20857.535} C_VEL
LIN {X 0,Y 323.567,Z 609.445,A -85,B 0,C 180,E1 20859.323,E2 20859.323} C_VEL
LIN {X 0,Y 318.469,Z 603.689,A -85,B 0,C 180,E1 20862.188,E2 20862.188} C_VEL
LIN {X 0,Y 318.149,Z 601.31,A -85,B 0,C 180,E1 20862.703,E2 20862.703} C_VEL
LIN {X 0,Y 318.677,Z 601.31,A -85,B 0,C 180,E1 20869.035,E2 20869.035} C_VEL
LIN {X 0,Y 319.464,Z 601.31,A -85,B 0,C 180,E1 20877.279,E2 20877.279} C_VEL
LIN {X 0,Y 319.497,Z 601.31,A -85,B 0,C 180,E1 20882.714,E2 20882.714} C_VEL
LIN {X 0,Y 318.706,Z 601.31,A -85,B 0,C 180,E1 20890.957,E2 20890.957} C_VEL
LIN {X 0,Y 318.066,Z 601.31,A -85,B 0,C 180,E1 20899.471,E2 20899.471} C_VEL
LIN {X 0,Y 318.025,Z 602.177,A -85,B 0,C 180,E1 20900.658,E2 20900.658} C_VEL
LIN {X 0,Y 321.009,Z 607.623,A -85,B 0,C 180,E1 20902.726,E2 20902.726} C_VEL
LIN {X 0,Y 323.125,Z 609.946,A -85,B 0,C 180,E1 20903.939,E2 20903.939} C_VEL
LIN {X 0,Y 327.095,Z 615.487,A -85,B 0,C 180,E1 20906.103,E2 20906.103} C_VEL
LIN {X 0,Y 340.221,Z 636.713,A -85,B 0,C 180,E1 20912.294,E2 20912.294} C_VEL
LIN {X 0,Y 354.358,Z 661.945,A -85,B 0,C 180,E1 20917.72,E2 20917.72} C_VEL
LIN {X 0,Y 367.516,Z 691.053,A -85,B 0,C 180,E1 20922.299,E2 20922.299} C_VEL
LIN {X 0,Y 376.168,Z 719.032,A -85,B 0,C 180,E1 20925.952,E2 20925.952} C_VEL
LIN {X 0,Y 376.384,Z 724.612,A -85,B 0,C 180,E1 20926.498,E2 20926.498} C_VEL
LIN {X 0,Y 368.271,Z 760.726,A -85,B 0,C 180,E1 20929.306,E2 20929.306} C_VEL
LIN {X 0,Y 358.617,Z 794.064,A -85,B 0,C 180,E1 20932.973,E2 20932.973} C_VEL
LIN {X 0,Y 348.581,Z 823.091,A -85,B 0,C 180,E1 20937.45,E2 20937.45} C_VEL
LIN {X 0,Y 339.19,Z 847.837,A -85,B 0,C 180,E1 20942.742,E2 20942.742} C_VEL
LIN {X 0,Y 331.692,Z 866.95,A -85,B 0,C 180,E1 20948.557,E2 20948.557} C_VEL
LIN {X 0,Y 326.259,Z 881.707,A -85,B 0,C 180,E1 20955.193,E2 20955.193} C_VEL
LIN {X 0,Y 323.303,Z 890.582,A -85,B 0,C 180,E1 20961.91,E2 20961.91} C_VEL
LIN {X 0,Y 322.484,Z 893.808,A -85,B 0,C 180,E1 20967.3,E2 20967.3} C_VEL
LIN {X 0,Y 322.587,Z 893.761,A -85,B 0,C 180,E1 20972.685,E2 20972.685} C_VEL
LIN {X 0,Y 323.79,Z 889.099,A -85,B 0,C 180,E1 20979.419,E2 20979.419} C_VEL
LIN {X 0,Y 327.205,Z 879.073,A -85,B 0,C 180,E1 20986.124,E2 20986.124} C_VEL
LIN {X 0,Y 333.224,Z 862.928,A -85,B 0,C 180,E1 20992.729,E2 20992.729} C_VEL
LIN {X 0,Y 341.29,Z 842.248,A -85,B 0,C 180,E1 20998.499,E2 20998.499} C_VEL
LIN {X 0,Y 351.164,Z 815.618,A -85,B 0,C 180,E1 21003.739,E2 21003.739} C_VEL
LIN {X 0,Y 361.244,Z 785.221,A -85,B 0,C 180,E1 21008.02,E2 21008.02} C_VEL
LIN {X 0,Y 370.52,Z 751.12,A -85,B 0,C 180,E1 21011.442,E2 21011.442} C_VEL
LIN {X 0,Y 376.595,Z 721.601,A -85,B 0,C 180,E1 21013.613,E2 21013.613} C_VEL
LIN {X 0,Y 369.002,Z 694.879,A -85,B 0,C 180,E1 21017.041,E2 21017.041} C_VEL
LIN {X 0,Y 355.644,Z 664.727,A -85,B 0,C 180,E1 21021.657,E2 21021.657} C_VEL
LIN {X 0,Y 350.498,Z 655.745,A -85,B 0,C 180,E1 21023.446,E2 21023.446} C_VEL
LIN {X 0,Y 341.556,Z 664.367,A -85,B 0,C 180,E1 21025.021,E2 21025.021} C_VEL
LIN {X 0,Y 340.644,Z 664.894,A -85,B 0,C 180,E1 21025.383,E2 21025.383} C_VEL
LIN {X 0,Y 348.203,Z 691.982,A -85,B 0,C 180,E1 21027.073,E2 21027.073} C_VEL
LIN {X 0,Y 343.483,Z 734.534,A -85,B 0,C 180,E1 21029.245,E2 21029.245} C_VEL
LIN {X 0,Y 337.792,Z 775.639,A -85,B 0,C 180,E1 21032.456,E2 21032.456} C_VEL
LIN {X 0,Y 332.407,Z 811.774,A -85,B 0,C 180,E1 21036.503,E2 21036.503} C_VEL
LIN {X 0,Y 327.993,Z 841.782,A -85,B 0,C 180,E1 21041.141,E2 21041.141} C_VEL
LIN {X 0,Y 324.722,Z 867.187,A -85,B 0,C 180,E1 21046.515,E2 21046.515} C_VEL
LIN {X 0,Y 323.084,Z 885.369,A -85,B 0,C 180,E1 21051.917,E2 21051.917} C_VEL
LIN {X 0,Y 322.892,Z 897.902,A -85,B 0,C 180,E1 21057.314,E2 21057.314} C_VEL
LIN {X 0,Y 323.568,Z 905.441,A -85,B 0,C 180,E1 21062.687,E2 21062.687} C_VEL
LIN {X 0,Y 326.305,Z 908.299,A -85,B 0,C 180,E1 21068.009,E2 21068.009} C_VEL
LIN {X 0,Y 330.617,Z 906.768,A -85,B 0,C 180,E1 21073.247,E2 21073.247} C_VEL
LIN {X 0,Y 338.159,Z 899.98,A -85,B 0,C 180,E1 21078.956,E2 21078.956} C_VEL
LIN {X 0,Y 350.182,Z 886.36,A -85,B 0,C 180,E1 21084.951,E2 21084.951} C_VEL
LIN {X 0,Y 368.529,Z 864.574,A -85,B 0,C 180,E1 21090.923,E2 21090.923} C_VEL
LIN {X 0,Y 391.566,Z 837.933,A -85,B 0,C 180,E1 21095.818,E2 21095.818} C_VEL
LIN {X 0,Y 400.565,Z 827.85,A -85,B 0,C 180,E1 21097.239,E2 21097.239} C_VEL
LIN {X 0,Y 401.878,Z 826.669,A -85,B 0,C 180,E1 21097.659,E2 21097.659} C_VEL
LIN {X 0,Y 374.546,Z 867.095,A -85,B 0,C 180,E1 21102.851,E2 21102.851} C_VEL
LIN {X 0,Y 352.37,Z 901.902,A -85,B 0,C 180,E1 21109.357,E2 21109.357} C_VEL
LIN {X 0,Y 336.336,Z 930.286,A -85,B 0,C 180,E1 21116.863,E2 21116.863} C_VEL
LIN {X 0,Y 326.771,Z 950.87,A -85,B 0,C 180,E1 21124.426,E2 21124.426} C_VEL
LIN {X 0,Y 322.148,Z 965.849,A -85,B 0,C 180,E1 21132.206,E2 21132.206} C_VEL
LIN {X 0,Y 320.929,Z 974.413,A -85,B 0,C 180,E1 21139.122,E2 21139.122} C_VEL
LIN {X 0,Y 321.152,Z 978.058,A -85,B 0,C 180,E1 21144.593,E2 21144.593} C_VEL
LIN {X 0,Y 321.812,Z 978.667,A -85,B 0,C 180,E1 21150.007,E2 21150.007} C_VEL
LIN {X 0,Y 321.441,Z 974.719,A -85,B 0,C 180,E1 21156.775,E2 21156.775} C_VEL
LIN {X 0,Y 321.704,Z 965.347,A -85,B 0,C 180,E1 21163.629,E2 21163.629} C_VEL
LIN {X 0,Y 323.76,Z 950.186,A -85,B 0,C 180,E1 21171.127,E2 21171.127} C_VEL
LIN {X 0,Y 328.363,Z 931.203,A -85,B 0,C 180,E1 21177.488,E2 21177.488} C_VEL
LIN {X 0,Y 335.057,Z 907.042,A -85,B 0,C 180,E1 21183.256,E2 21183.256} C_VEL
LIN {X 0,Y 343.148,Z 878.251,A -85,B 0,C 180,E1 21188.192,E2 21188.192} C_VEL
LIN {X 0,Y 351.292,Z 845.813,A -85,B 0,C 180,E1 21192.173,E2 21192.173} C_VEL
LIN {X 0,Y 361.326,Z 806.889,A -85,B 0,C 180,E1 21196.119,E2 21196.119} C_VEL
LIN {X 0,Y 370.583,Z 764.499,A -85,B 0,C 180,E1 21199.185,E2 21199.185} C_VEL
LIN {X 0,Y 375.432,Z 733.691,A -85,B 0,C 180,E1 21200.845,E2 21200.845} C_VEL
LIN {X 0,Y 362.669,Z 701.584,A -85,B 0,C 180,E1 21203.634,E2 21203.634} C_VEL
LIN {X 0,Y 357.068,Z 692.438,A -85,B 0,C 180,E1 21204.84,E2 21204.84} C_VEL
LIN {X 0,Y 349.081,Z 680.258,A -85,B 0,C 180,E1 21207.031,E2 21207.031} C_VEL
LIN {X 0,Y 348.573,Z 678.553,A -85,B 0,C 180,E1 21207.243,E2 21207.243} C_VEL
LIN {X 0,Y 338.791,Z 642.139,A -85,B 0,C 180,E1 21211.904,E2 21211.904} C_VEL
LIN {X 0,Y 327.952,Z 626.952,A -85,B 0,C 180,E1 21216.427,E2 21216.427} C_VEL
LIN {X 0,Y 324.274,Z 621.711,A -85,B 0,C 180,E1 21218.231,E2 21218.231} C_VEL
LIN {X 0,Y 320.027,Z 615.517,A -85,B 0,C 180,E1 21220.556,E2 21220.556} C_VEL
LIN {X 0,Y 316.121,Z 609.759,A -85,B 0,C 180,E1 21222.996,E2 21222.996} C_VEL
LIN {X 0,Y 310.9,Z 603.663,A -85,B 0,C 180,E1 21226.846,E2 21226.846} C_VEL
LIN {X 0,Y 310.553,Z 601.31,A -85,B 0,C 180,E1 21227.408,E2 21227.408} C_VEL
LIN {X 0,Y 311.306,Z 601.31,A -85,B 0,C 180,E1 21234.411,E2 21234.411} C_VEL
LIN {X 0,Y 311.866,Z 601.31,A -85,B 0,C 180,E1 21239.996,E2 21239.996} C_VEL
LIN {X 0,Y 311.006,Z 601.31,A -85,B 0,C 180,E1 21248.399,E2 21248.399} C_VEL
LIN {X 0,Y 310.413,Z 602.101,A -85,B 0,C 180,E1 21255.929,E2 21255.929} C_VEL
LIN {X 0,Y 313.083,Z 607.414,A -85,B 0,C 180,E1 21258.451,E2 21258.451} C_VEL
LIN {X 0,Y 315.681,Z 609.959,A -85,B 0,C 180,E1 21260.264,E2 21260.264} C_VEL
LIN {X 0,Y 319.625,Z 615.657,A -85,B 0,C 180,E1 21262.929,E2 21262.929} C_VEL
LIN {X 0,Y 329.369,Z 631.13,A -85,B 0,C 180,E1 21268.377,E2 21268.377} C_VEL
LIN {X 0,Y 340.896,Z 650.442,A -85,B 0,C 180,E1 21273.549,E2 21273.549} C_VEL
LIN {X 0,Y 353.481,Z 674.708,A -85,B 0,C 180,E1 21278.427,E2 21278.427} C_VEL
LIN {X 0,Y 365.418,Z 704.093,A -85,B 0,C 180,E1 21282.862,E2 21282.862} C_VEL
LIN {X 0,Y 370.654,Z 725.928,A -85,B 0,C 180,E1 21285.687,E2 21285.687} C_VEL
LIN {X 0,Y 362.442,Z 761.503,A -85,B 0,C 180,E1 21288.476,E2 21288.476} C_VEL
LIN {X 0,Y 352.76,Z 793.901,A -85,B 0,C 180,E1 21292.057,E2 21292.057} C_VEL
LIN {X 0,Y 342.626,Z 822.453,A -85,B 0,C 180,E1 21296.433,E2 21296.433} C_VEL
LIN {X 0,Y 332.756,Z 847.555,A -85,B 0,C 180,E1 21301.8,E2 21301.8} C_VEL
LIN {X 0,Y 324.365,Z 867.975,A -85,B 0,C 180,E1 21308.048,E2 21308.048} C_VEL
LIN {X 0,Y 318.644,Z 882.708,A -85,B 0,C 180,E1 21314.831,E2 21314.831} C_VEL
LIN {X 0,Y 315.546,Z 891.576,A -85,B 0,C 180,E1 21321.71,E2 21321.71} C_VEL
LIN {X 0,Y 314.669,Z 894.794,A -85,B 0,C 180,E1 21327.232,E2 21327.232} C_VEL
LIN {X 0,Y 314.762,Z 894.749,A -85,B 0,C 180,E1 21332.752,E2 21332.752} C_VEL
LIN {X 0,Y 316.047,Z 890.099,A -85,B 0,C 180,E1 21339.652,E2 21339.652} C_VEL
LIN {X 0,Y 319.65,Z 880.086,A -85,B 0,C 180,E1 21346.516,E2 21346.516} C_VEL
LIN {X 0,Y 325.965,Z 863.944,A -85,B 0,C 180,E1 21353.265,E2 21353.265} C_VEL
LIN {X 0,Y 334.403,Z 843.29,A -85,B 0,C 180,E1 21359.141,E2 21359.141} C_VEL
LIN {X 0,Y 344.677,Z 816.668,A -85,B 0,C 180,E1 21364.462,E2 21364.462} C_VEL
LIN {X 0,Y 355.088,Z 786.244,A -85,B 0,C 180,E1 21368.801,E2 21368.801} C_VEL
LIN {X 0,Y 364.525,Z 752.732,A -85,B 0,C 180,E1 21372.203,E2 21372.203} C_VEL
LIN {X 0,Y 370.501,Z 723.65,A -85,B 0,C 180,E1 21374.422,E2 21374.422} C_VEL
LIN {X 0,Y 363.162,Z 697.626,A -85,B 0,C 180,E1 21377.908,E2 21377.908} C_VEL
LIN {X 0,Y 350.521,Z 668.769,A -85,B 0,C 180,E1 21382.51,E2 21382.51} C_VEL
LIN {X 0,Y 348.364,Z 665.513,A -85,B 0,C 180,E1 21383.25,E2 21383.25} C_VEL
LIN {X 0,Y 340.447,Z 673.652,A -85,B 0,C 180,E1 21384.573,E2 21384.573} C_VEL
LIN {X 0,Y 337.401,Z 676.101,A -85,B 0,C 180,E1 21385.165,E2 21385.165} C_VEL
LIN {X 0,Y 336.49,Z 676.322,A -85,B 0,C 180,E1 21385.487,E2 21385.487} C_VEL
LIN {X 0,Y 341.003,Z 692.146,A -85,B 0,C 180,E1 21386.541,E2 21386.541} C_VEL
LIN {X 0,Y 336.05,Z 735.788,A -85,B 0,C 180,E1 21388.827,E2 21388.827} C_VEL
LIN {X 0,Y 330.407,Z 775.319,A -85,B 0,C 180,E1 21391.973,E2 21391.973} C_VEL
LIN {X 0,Y 324.837,Z 811.614,A -85,B 0,C 180,E1 21396.104,E2 21396.104} C_VEL
LIN {X 0,Y 320.185,Z 842.532,A -85,B 0,C 180,E1 21400.963,E2 21400.963} C_VEL
LIN {X 0,Y 316.953,Z 866.87,A -85,B 0,C 180,E1 21406.177,E2 21406.177} C_VEL
LIN {X 0,Y 315.236,Z 885.493,A -85,B 0,C 180,E1 21411.714,E2 21411.714} C_VEL
LIN {X 0,Y 315.032,Z 898.382,A -85,B 0,C 180,E1 21417.247,E2 21417.247} C_VEL
LIN {X 0,Y 315.725,Z 906.282,A -85,B 0,C 180,E1 21422.754,E2 21422.754} C_VEL
LIN {X 0,Y 318.578,Z 909.543,A -85,B 0,C 180,E1 21428.205,E2 21428.205} C_VEL
LIN {X 0,Y 323.129,Z 908.464,A -85,B 0,C 180,E1 21433.56,E2 21433.56} C_VEL
LIN {X 0,Y 332.085,Z 901.286,A -85,B 0,C 180,E1 21440.01,E2 21440.01} C_VEL
LIN {X 0,Y 345.119,Z 887.918,A -85,B 0,C 180,E1 21446.04,E2 21446.04} C_VEL
LIN {X 0,Y 364.675,Z 866.895,A -85,B 0,C 180,E1 21451.985,E2 21451.985} C_VEL
LIN {X 0,Y 389.486,Z 840.82,A -85,B 0,C 180,E1 21456.875,E2 21456.875} C_VEL
LIN {X 0,Y 392.984,Z 837.304,A -85,B 0,C 180,E1 21457.403,E2 21457.403} C_VEL
LIN {X 0,Y 386.369,Z 846.391,A -85,B 0,C 180,E1 21458.687,E2 21458.687} C_VEL
LIN {X 0,Y 360.912,Z 881.672,A -85,B 0,C 180,E1 21464.107,E2 21464.107} C_VEL
LIN {X 0,Y 339.277,Z 914.205,A -85,B 0,C 180,E1 21471.309,E2 21471.309} C_VEL
LIN {X 0,Y 324.823,Z 939.222,A -85,B 0,C 180,E1 21479.137,E2 21479.137} C_VEL
LIN {X 0,Y 316.517,Z 958.026,A -85,B 0,C 180,E1 21487.49,E2 21487.49} C_VEL
LIN {X 0,Y 313.324,Z 970.691,A -85,B 0,C 180,E1 21496.015,E2 21496.015} C_VEL
LIN {X 0,Y 313.107,Z 975.643,A -85,B 0,C 180,E1 21501.66,E2 21501.66} C_VEL
LIN {X 0,Y 313.641,Z 977.658,A -85,B 0,C 180,E1 21507.239,E2 21507.239} C_VEL
LIN {X 0,Y 314.018,Z 977.503,A -85,B 0,C 180,E1 21510.008,E2 21510.008} C_VEL
LIN {X 0,Y 313.647,Z 973.586,A -85,B 0,C 180,E1 21516.722,E2 21516.722} C_VEL
LIN {X 0,Y 313.964,Z 963.093,A -85,B 0,C 180,E1 21524.608,E2 21524.608} C_VEL
LIN {X 0,Y 316.207,Z 948.856,A -85,B 0,C 180,E1 21531.758,E2 21531.758} C_VEL
LIN {X 0,Y 321.416,Z 928.532,A -85,B 0,C 180,E1 21538.606,E2 21538.606} C_VEL
LIN {X 0,Y 328.642,Z 904.145,A -85,B 0,C 180,E1 21544.396,E2 21544.396} C_VEL
LIN {X 0,Y 337.027,Z 875.562,A -85,B 0,C 180,E1 21549.28,E2 21549.28} C_VEL
LIN {X 0,Y 345.424,Z 843.5,A -85,B 0,C 180,E1 21553.2,E2 21553.2} C_VEL
LIN {X 0,Y 359.092,Z 785.141,A -85,B 0,C 180,E1 21558.355,E2 21558.355} C_VEL
LIN {X 0,Y 367.892,Z 741.717,A -85,B 0,C 180,E1 21560.987,E2 21560.987} C_VEL
LIN {X 0,Y 368.234,Z 735.812,A -85,B 0,C 180,E1 21561.329,E2 21561.329} C_VEL
LIN {X 0,Y 353.944,Z 698.35,A -85,B 0,C 180,E1 21564.855,E2 21564.855} C_VEL
LIN {X 0,Y 348.573,Z 678.553,A -85,B 0,C 180,E1 21567.243,E2 21567.243} C_VEL
LIN {X 0,Y 346.134,Z 672.394,A -85,B 0,C 180,E1 21568.184,E2 21568.184} C_VEL
LIN {X 0,Y 338.101,Z 658.086,A -85,B 0,C 180,E1 21571.179,E2 21571.179} C_VEL
LIN {X 0,Y 337.651,Z 656.438,A -85,B 0,C 180,E1 21571.414,E2 21571.414} C_VEL
LIN {X 0,Y 335.156,Z 648.045,A -85,B 0,C 180,E1 21572.67,E2 21572.67} C_VEL
LIN {X 0,Y 322.703,Z 629.63,A -85,B 0,C 180,E1 21578.3,E2 21578.3} C_VEL
LIN {X 0,Y 317.466,Z 622.518,A -85,B 0,C 180,E1 21581.207,E2 21581.207} C_VEL
LIN {X 0,Y 312.98,Z 615.965,A -85,B 0,C 180,E1 21584.198,E2 21584.198} C_VEL
LIN {X 0,Y 308.958,Z 610.629,A -85,B 0,C 180,E1 21587.426,E2 21587.426} C_VEL
LIN {X 0,Y 308.098,Z 608.788,A -85,B 0,C 180,E1 21588.317,E2 21588.317} C_VEL
LIN {X 0,Y 303.617,Z 603.599,A -85,B 0,C 180,E1 21593.73,E2 21593.73} C_VEL
LIN {X 0,Y 303.411,Z 601.31,A -85,B 0,C 180,E1 21595.056,E2 21595.056} C_VEL
LIN {X 0,Y 303.959,Z 601.31,A -85,B 0,C 180,E1 21599.996,E2 21599.996} C_VEL
LIN {X 0,Y 303.133,Z 601.859,A -85,B 0,C 180,E1 21608.438,E2 21608.438} C_VEL
LIN {X 0,Y 304.845,Z 606.642,A -85,B 0,C 180,E1 21611.819,E2 21611.819} C_VEL
LIN {X 0,Y 308.369,Z 609.957,A -85,B 0,C 180,E1 21615.581,E2 21615.581} C_VEL
LIN {X 0,Y 311.871,Z 615.542,A -85,B 0,C 180,E1 21618.768,E2 21618.768} C_VEL
LIN {X 0,Y 313.588,Z 618.101,A -85,B 0,C 180,E1 21620.123,E2 21620.123} C_VEL
LIN {X 0,Y 318.623,Z 625.888,A -85,B 0,C 180,E1 21623.544,E2 21623.544} C_VEL
LIN {X 0,Y 326.277,Z 637.775,A -85,B 0,C 180,E1 21627.859,E2 21627.859} C_VEL
LIN {X 0,Y 338.585,Z 659.058,A -85,B 0,C 180,E1 21633.616,E2 21633.616} C_VEL
LIN {X 0,Y 351.672,Z 685.998,A -85,B 0,C 180,E1 21638.842,E2 21638.842} C_VEL
LIN {X 0,Y 361.443,Z 712.8,A -85,B 0,C 180,E1 21642.845,E2 21642.845} C_VEL
LIN {X 0,Y 364.698,Z 728.838,A -85,B 0,C 180,E1 21644.954,E2 21644.954} C_VEL
LIN {X 0,Y 355.785,Z 765.448,A -85,B 0,C 180,E1 21647.923,E2 21647.923} C_VEL
LIN {X 0,Y 345.445,Z 798.319,A -85,B 0,C 180,E1 21651.708,E2 21651.708} C_VEL
LIN {X 0,Y 334.777,Z 826.825,A -85,B 0,C 180,E1 21656.319,E2 21656.319} C_VEL
LIN {X 0,Y 324.753,Z 851.102,A -85,B 0,C 180,E1 21661.801,E2 21661.801} C_VEL
LIN {X 0,Y 316.491,Z 870.299,A -85,B 0,C 180,E1 21668.022,E2 21668.022} C_VEL
LIN {X 0,Y 310.633,Z 884.861,A -85,B 0,C 180,E1 21675.154,E2 21675.154} C_VEL
LIN {X 0,Y 307.775,Z 892.572,A -85,B 0,C 180,E1 21681.499,E2 21681.499} C_VEL
LIN {X 0,Y 306.848,Z 895.781,A -85,B 0,C 180,E1 21687.162,E2 21687.162} C_VEL
LIN {X 0,Y 306.94,Z 895.737,A -85,B 0,C 180,E1 21692.822,E2 21692.822} C_VEL
LIN {X 0,Y 308.296,Z 891.176,A -85,B 0,C 180,E1 21699.812,E2 21699.812} C_VEL
LIN {X 0,Y 312.093,Z 881.101,A -85,B 0,C 180,E1 21706.928,E2 21706.928} C_VEL
LIN {X 0,Y 318.74,Z 864.978,A -85,B 0,C 180,E1 21713.824,E2 21713.824} C_VEL
LIN {X 0,Y 327.544,Z 844.337,A -85,B 0,C 180,E1 21719.812,E2 21719.812} C_VEL
LIN {X 0,Y 338.244,Z 817.697,A -85,B 0,C 180,E1 21725.214,E2 21725.214} C_VEL
LIN {X 0,Y 349.002,Z 787.271,A -85,B 0,C 180,E1 21729.609,E2 21729.609} C_VEL
LIN {X 0,Y 358.933,Z 753.14,A -85,B 0,C 180,E1 21733.096,E2 21733.096} C_VEL
LIN {X 0,Y 364.526,Z 725.897,A -85,B 0,C 180,E1 21735.232,E2 21735.232} C_VEL
LIN {X 0,Y 357.112,Z 699.577,A -85,B 0,C 180,E1 21738.923,E2 21738.923} C_VEL
LIN {X 0,Y 346.355,Z 675.217,A -85,B 0,C 180,E1 21743.002,E2 21743.002} C_VEL
LIN {X 0,Y 333.419,Z 687.561,A -85,B 0,C 180,E1 21745.251,E2 21745.251} C_VEL
LIN {X 0,Y 332.318,Z 687.947,A -85,B 0,C 180,E1 21745.647,E2 21745.647} C_VEL
LIN {X 0,Y 333.45,Z 695.932,A -85,B 0,C 180,E1 21746.132,E2 21746.132} C_VEL
LIN {X 0,Y 328.208,Z 739.801,A -85,B 0,C 180,E1 21748.571,E2 21748.571} C_VEL
LIN {X 0,Y 322.282,Z 779.848,A -85,B 0,C 180,E1 21751.966,E2 21751.966} C_VEL
LIN {X 0,Y 316.513,Z 816.383,A -85,B 0,C 180,E1 21756.373,E2 21756.373} C_VEL
LIN {X 0,Y 311.79,Z 847.296,A -85,B 0,C 180,E1 21761.545,E2 21761.545} C_VEL
LIN {X 0,Y 308.593,Z 871.805,A -85,B 0,C 180,E1 21767.241,E2 21767.241} C_VEL
LIN {X 0,Y 307.198,Z 889.439,A -85,B 0,C 180,E1 21772.922,E2 21772.922} C_VEL
LIN {X 0,Y 307.159,Z 901.382,A -85,B 0,C 180,E1 21778.591,E2 21778.591} C_VEL
LIN {X 0,Y 308.449,Z 908.48,A -85,B 0,C 180,E1 21784.228,E2 21784.228} C_VEL
LIN {X 0,Y 310.872,Z 910.778,A -85,B 0,C 180,E1 21788.41,E2 21788.41} C_VEL
LIN {X 0,Y 315.637,Z 910.181,A -85,B 0,C 180,E1 21793.888,E2 21793.888} C_VEL
LIN {X 0,Y 325.03,Z 903.614,A -85,B 0,C 180,E1 21800.464,E2 21800.464} C_VEL
LIN {X 0,Y 338.62,Z 891.222,A -85,B 0,C 180,E1 21806.579,E2 21806.579} C_VEL
LIN {X 0,Y 358.873,Z 871.399,A -85,B 0,C 180,E1 21812.565,E2 21812.565} C_VEL
LIN {X 0,Y 383.869,Z 847.567,A -85,B 0,C 180,E1 21817.363,E2 21817.363} C_VEL
LIN {X 0,Y 375.361,Z 858.372,A -85,B 0,C 180,E1 21818.999,E2 21818.999} C_VEL
LIN {X 0,Y 349.74,Z 891.558,A -85,B 0,C 180,E1 21824.822,E2 21824.822} C_VEL
LIN {X 0,Y 328.326,Z 921.886,A -85,B 0,C 180,E1 21832.457,E2 21832.457} C_VEL
LIN {X 0,Y 314.204,Z 945.903,A -85,B 0,C 180,E1 21841.177,E2 21841.177} C_VEL
LIN {X 0,Y 307.262,Z 962.331,A -85,B 0,C 180,E1 21849.815,E2 21849.815} C_VEL
LIN {X 0,Y 305.311,Z 971.321,A -85,B 0,C 180,E1 21857.104,E2 21857.104} C_VEL
LIN {X 0,Y 305.451,Z 975.994,A -85,B 0,C 180,E1 21864.314,E2 21864.314} C_VEL
LIN {X 0,Y 306.197,Z 976.32,A -85,B 0,C 180,E1 21870.008,E2 21870.008} C_VEL
LIN {X 0,Y 305.861,Z 973.215,A -85,B 0,C 180,E1 21875.694,E2 21875.694} C_VEL
LIN {X 0,Y 305.971,Z 964.051,A -85,B 0,C 180,E1 21883.613,E2 21883.613} C_VEL
LIN {X 0,Y 307.889,Z 950.581,A -85,B 0,C 180,E1 21891.098,E2 21891.098} C_VEL
LIN {X 0,Y 313.027,Z 931.315,A -85,B 0,C 180,E1 21898.169,E2 21898.169} C_VEL
LIN {X 0,Y 320.392,Z 907.461,A -85,B 0,C 180,E1 21904.288,E2 21904.288} C_VEL
LIN {X 0,Y 329.099,Z 879.552,A -85,B 0,C 180,E1 21909.403,E2 21909.403} C_VEL
LIN {X 0,Y 338.105,Z 847.549,A -85,B 0,C 180,E1 21913.585,E2 21913.585} C_VEL
LIN {X 0,Y 345.909,Z 813.097,A -85,B 0,C 180,E1 21916.749,E2 21916.749} C_VEL
LIN {X 0,Y 358.005,Z 757.258,A -85,B 0,C 180,E1 21920.73,E2 21920.73} C_VEL
LIN {X 0,Y 361.196,Z 738.316,A -85,B 0,C 180,E1 21921.783,E2 21921.783} C_VEL
LIN {X 0,Y 351.956,Z 713.039,A -85,B 0,C 180,E1 21924.308,E2 21924.308} C_VEL
LIN {X 0,Y 337.651,Z 656.438,A -85,B 0,C 180,E1 21931.414,E2 21931.414} C_VEL
LIN {X 0,Y 334.648,Z 652.174,A -85,B 0,C 180,E1 21932.582,E2 21932.582} C_VEL
LIN {X 0,Y 328.188,Z 648.617,A -85,B 0,C 180,E1 21934.904,E2 21934.904} C_VEL
LIN {X 0,Y 318.671,Z 634.714,A -85,B 0,C 180,E1 21939.655,E2 21939.655} C_VEL
LIN {X 0,Y 315.242,Z 629.64,A -85,B 0,C 180,E1 21941.705,E2 21941.705} C_VEL
LIN {X 0,Y 310.744,Z 623.267,A -85,B 0,C 180,E1 21944.806,E2 21944.806} C_VEL
LIN {X 0,Y 306.917,Z 617.188,A -85,B 0,C 180,E1 21948.158,E2 21948.158} C_VEL
LIN {X 0,Y 302.065,Z 610.736,A -85,B 0,C 180,E1 21954.33,E2 21954.33} C_VEL
LIN {X 0,Y 301.543,Z 608.98,A -85,B 0,C 180,E1 21955.675,E2 21955.675} C_VEL
LIN {X 0,Y 300.863,Z 608.841,A -85,B 0,C 180,E1 21966.501,E2 21966.501} C_VEL
LIN {X 0,Y 301.535,Z 610.14,A -85,B 0,C 180,E1 21968.301,E2 21968.301} C_VEL
LIN {X 0,Y 304.692,Z 615.689,A -85,B 0,C 180,E1 21973.473,E2 21973.473} C_VEL
LIN {X 0,Y 306.458,Z 617.705,A -85,B 0,C 180,E1 21975.313,E2 21975.313} C_VEL
LIN {X 0,Y 310.28,Z 623.37,A -85,B 0,C 180,E1 21978.874,E2 21978.874} C_VEL
LIN {X 0,Y 319.179,Z 637.753,A -85,B 0,C 180,E1 21985.088,E2 21985.088} C_VEL
LIN {X 0,Y 330.406,Z 657.167,A -85,B 0,C 180,E1 21991.047,E2 21991.047} C_VEL
LIN {X 0,Y 342.631,Z 681.09,A -85,B 0,C 180,E1 21996.401,E2 21996.401} C_VEL
LIN {X 0,Y 353.628,Z 708.702,A -85,B 0,C 180,E1 22000.988,E2 22000.988} C_VEL
LIN {X 0,Y 358.991,Z 730.833,A -85,B 0,C 180,E1 22004.14,E2 22004.14} C_VEL
LIN {X 0,Y 350.029,Z 766.382,A -85,B 0,C 180,E1 22007.058,E2 22007.058} C_VEL
LIN {X 0,Y 339.34,Z 799.372,A -85,B 0,C 180,E1 22010.889,E2 22010.889} C_VEL
LIN {X 0,Y 328.267,Z 827.875,A -85,B 0,C 180,E1 22015.559,E2 22015.559} C_VEL
LIN {X 0,Y 317.843,Z 852.141,A -85,B 0,C 180,E1 22021.131,E2 22021.131} C_VEL
LIN {X 0,Y 309.003,Z 871.766,A -85,B 0,C 180,E1 22027.657,E2 22027.657} C_VEL
LIN {X 0,Y 303.019,Z 885.869,A -85,B 0,C 180,E1 22034.772,E2 22034.772} C_VEL
LIN {X 0,Y 300.015,Z 893.566,A -85,B 0,C 180,E1 22041.277,E2 22041.277} C_VEL
LIN {X 0,Y 299.014,Z 896.771,A -85,B 0,C 180,E1 22047.087,E2 22047.087} C_VEL
LIN {X 0,Y 299.128,Z 896.723,A -85,B 0,C 180,E1 22052.896,E2 22052.896} C_VEL
LIN {X 0,Y 300.448,Z 892.467,A -85,B 0,C 180,E1 22059.769,E2 22059.769} C_VEL
LIN {X 0,Y 304.566,Z 882.116,A -85,B 0,C 180,E1 22067.359,E2 22067.359} C_VEL
LIN {X 0,Y 311.538,Z 866.011,A -85,B 0,C 180,E1 22074.411,E2 22074.411} C_VEL
LIN {X 0,Y 320.739,Z 845.383,A -85,B 0,C 180,E1 22080.511,E2 22080.511} C_VEL
LIN {X 0,Y 331.857,Z 818.738,A -85,B 0,C 180,E1 22085.996,E2 22085.996} C_VEL
LIN {X 0,Y 342.988,Z 788.311,A -85,B 0,C 180,E1 22090.445,E2 22090.445} C_VEL
LIN {X 0,Y 353.305,Z 754.004,A -85,B 0,C 180,E1 22093.979,E2 22093.979} C_VEL
LIN {X 0,Y 358.847,Z 729.69,A -85,B 0,C 180,E1 22095.865,E2 22095.865} C_VEL
LIN {X 0,Y 351.872,Z 703.433,A -85,B 0,C 180,E1 22099.679,E2 22099.679} C_VEL
LIN {X 0,Y 343.994,Z 684.951,A -85,B 0,C 180,E1 22102.817,E2 22102.817} C_VEL
LIN {X 0,Y 332.232,Z 696.553,A -85,B 0,C 180,E1 22104.783,E2 22104.783} C_VEL
LIN {X 0,Y 326.75,Z 704.196,A -85,B 0,C 180,E1 22105.564,E2 22105.564} C_VEL
LIN {X 0,Y 325.398,Z 704.305,A -85,B 0,C 180,E1 22105.927,E2 22105.927} C_VEL
LIN {X 0,Y 319.71,Z 748.272,A -85,B 0,C 180,E1 22108.69,E2 22108.69} C_VEL
LIN {X 0,Y 313.658,Z 787.285,A -85,B 0,C 180,E1 22112.303,E2 22112.303} C_VEL
LIN {X 0,Y 308.042,Z 822.105,A -85,B 0,C 180,E1 22116.836,E2 22116.836} C_VEL
LIN {X 0,Y 303.358,Z 851.962,A -85,B 0,C 180,E1 22122.212,E2 22122.212} C_VEL
LIN {X 0,Y 300.413,Z 875.442,A -85,B 0,C 180,E1 22127.998,E2 22127.998} C_VEL
LIN {X 0,Y 299.198,Z 893.068,A -85,B 0,C 180,E1 22134.192,E2 22134.192} C_VEL
LIN {X 0,Y 299.476,Z 904.135,A -85,B 0,C 180,E1 22140.004,E2 22140.004} C_VEL
LIN {X 0,Y 301.372,Z 910.462,A -85,B 0,C 180,E1 22145.773,E2 22145.773} C_VEL
LIN {X 0,Y 305.355,Z 912.383,A -85,B 0,C 180,E1 22151.45,E2 22151.45} C_VEL
LIN {X 0,Y 313.493,Z 909.064,A -85,B 0,C 180,E1 22158.31,E2 22158.31} C_VEL
LIN {X 0,Y 325.902,Z 899.688,A -85,B 0,C 180,E1 22164.734,E2 22164.734} C_VEL
LIN {X 0,Y 344.86,Z 883.283,A -85,B 0,C 180,E1 22171.078,E2 22171.078} C_VEL
LIN {X 0,Y 370.8,Z 860.411,A -85,B 0,C 180,E1 22176.694,E2 22176.694} C_VEL
LIN {X 0,Y 374.752,Z 857.046,A -85,B 0,C 180,E1 22177.33,E2 22177.33} C_VEL
LIN {X 0,Y 343.328,Z 894.449,A -85,B 0,C 180,E1 22184.19,E2 22184.19} C_VEL
LIN {X 0,Y 321.816,Z 922.586,A -85,B 0,C 180,E1 22191.647,E2 22191.647} C_VEL
LIN {X 0,Y 307.019,Z 945.671,A -85,B 0,C 180,E1 22200.437,E2 22200.437} C_VEL
LIN {X 0,Y 299.61,Z 961.657,A -85,B 0,C 180,E1 22209.276,E2 22209.276} C_VEL
LIN {X 0,Y 297.321,Z 971.756,A -85,B 0,C 180,E1 22218.246,E2 22218.246} C_VEL
LIN {X 0,Y 297.578,Z 974.952,A -85,B 0,C 180,E1 22224.163,E2 22224.163} C_VEL
LIN {X 0,Y 298.376,Z 975.124,A -85,B 0,C 180,E1 22230.008,E2 22230.008} C_VEL
LIN {X 0,Y 297.958,Z 970.327,A -85,B 0,C 180,E1 22237.432,E2 22237.432} C_VEL
LIN {X 0,Y 298.29,Z 961.282,A -85,B 0,C 180,E1 22245.206,E2 22245.206} C_VEL
LIN {X 0,Y 301.023,Z 946.515,A -85,B 0,C 180,E1 22252.969,E2 22252.969} C_VEL
LIN {X 0,Y 306.439,Z 927.717,A -85,B 0,C 180,E1 22259.643,E2 22259.643} C_VEL
LIN {X 0,Y 314.506,Z 903.366,A -85,B 0,C 180,E1 22265.752,E2 22265.752} C_VEL
LIN {X 0,Y 323.897,Z 874.445,A -85,B 0,C 180,E1 22270.924,E2 22270.924} C_VEL
LIN {X 0,Y 333.118,Z 842.221,A -85,B 0,C 180,E1 22275.009,E2 22275.009} C_VEL
LIN {X 0,Y 341.455,Z 806.072,A -85,B 0,C 180,E1 22278.182,E2 22278.182} C_VEL
LIN {X 0,Y 353.995,Z 740.526,A -85,B 0,C 180,E1 22282.257,E2 22282.257} C_VEL
LIN {X 0,Y 347.331,Z 718.468,A -85,B 0,C 180,E1 22284.885,E2 22284.885} C_VEL
LIN {X 0,Y 332.042,Z 654.585,A -85,B 0,C 180,E1 22293.219,E2 22293.219} C_VEL
LIN {X 0,Y 328.188,Z 648.617,A -85,B 0,C 180,E1 22294.904,E2 22294.904} C_VEL
LIN {X 0,Y 323.258,Z 647.025,A -85,B 0,C 180,E1 22296.792,E2 22296.792} C_VEL
LIN {X 0,Y 318.814,Z 645.104,A -85,B 0,C 180,E1 22298.71,E2 22298.71} C_VEL
LIN {X 0,Y 312.026,Z 635.64,A -85,B 0,C 180,E1 22302.788,E2 22302.788} C_VEL
LIN {X 0,Y 308.697,Z 630.643,A -85,B 0,C 180,E1 22305.248,E2 22305.248} C_VEL
LIN {X 0,Y 304.406,Z 623.894,A -85,B 0,C 180,E1 22309.241,E2 22309.241} C_VEL
LIN {X 0,Y 300.416,Z 618.135,A -85,B 0,C 180,E1 22314.752,E2 22314.752} C_VEL
LIN {X 0,Y 299.752,Z 616.631,A -85,B 0,C 180,E1 22316.374,E2 22316.374} C_VEL
LIN {X 0,Y 299.778,Z 616.773,A -85,B 0,C 180,E1 22327.528,E2 22327.528} C_VEL
LIN {X 0,Y 301.818,Z 622.363,A -85,B 0,C 180,E1 22331.945,E2 22331.945} C_VEL
LIN {X 0,Y 304.415,Z 625.347,A -85,B 0,C 180,E1 22335.049,E2 22335.049} C_VEL
LIN {X 0,Y 309.229,Z 633.297,A -85,B 0,C 180,E1 22339.587,E2 22339.587} C_VEL
LIN {X 0,Y 316.466,Z 644.884,A -85,B 0,C 180,E1 22344.684,E2 22344.684} C_VEL
LIN {X 0,Y 326.926,Z 663.621,A -85,B 0,C 180,E1 22350.544,E2 22350.544} C_VEL
LIN {X 0,Y 338.76,Z 687.59,A -85,B 0,C 180,E1 22355.974,E2 22355.974} C_VEL
LIN {X 0,Y 348.744,Z 713.99,A -85,B 0,C 180,E1 22360.451,E2 22360.451} C_VEL
LIN {X 0,Y 353.051,Z 734.201,A -85,B 0,C 180,E1 22363.393,E2 22363.393} C_VEL
LIN {X 0,Y 343.778,Z 769.309,A -85,B 0,C 180,E1 22366.359,E2 22366.359} C_VEL
LIN {X 0,Y 332.444,Z 802.537,A -85,B 0,C 180,E1 22370.341,E2 22370.341} C_VEL
LIN {X 0,Y 321.114,Z 830.569,A -85,B 0,C 180,E1 22375.092,E2 22375.092} C_VEL
LIN {X 0,Y 310.394,Z 854.355,A -85,B 0,C 180,E1 22380.772,E2 22380.772} C_VEL
LIN {X 0,Y 301.742,Z 872.781,A -85,B 0,C 180,E1 22387.089,E2 22387.089} C_VEL
LIN {X 0,Y 295.433,Z 886.878,A -85,B 0,C 180,E1 22394.371,E2 22394.371} C_VEL
LIN {X 0,Y 292.259,Z 894.563,A -85,B 0,C 180,E1 22401.044,E2 22401.044} C_VEL
LIN {X 0,Y 291.194,Z 897.758,A -85,B 0,C 180,E1 22407.009,E2 22407.009} C_VEL
LIN {X 0,Y 291.306,Z 897.713,A -85,B 0,C 180,E1 22412.973,E2 22412.973} C_VEL
LIN {X 0,Y 292.942,Z 892.793,A -85,B 0,C 180,E1 22420.742,E2 22420.742} C_VEL
LIN {X 0,Y 297.572,Z 881.862,A -85,B 0,C 180,E1 22428.499,E2 22428.499} C_VEL
LIN {X 0,Y 305.309,Z 865.093,A -85,B 0,C 180,E1 22435.729,E2 22435.729} C_VEL
LIN {X 0,Y 315.194,Z 843.647,A -85,B 0,C 180,E1 22441.915,E2 22441.915} C_VEL
LIN {X 0,Y 326.731,Z 816.808,A -85,B 0,C 180,E1 22447.341,E2 22447.341} C_VEL
LIN {X 0,Y 338.347,Z 785.619,A -85,B 0,C 180,E1 22451.76,E2 22451.76} C_VEL
LIN {X 0,Y 348.742,Z 751.089,A -85,B 0,C 180,E1 22455.208,E2 22455.208} C_VEL
LIN {X 0,Y 353.05,Z 732.536,A -85,B 0,C 180,E1 22456.648,E2 22456.648} C_VEL
LIN {X 0,Y 346.243,Z 706.343,A -85,B 0,C 180,E1 22460.628,E2 22460.628} C_VEL
LIN {X 0,Y 341.566,Z 694.819,A -85,B 0,C 180,E1 22462.617,E2 22462.617} C_VEL
LIN {X 0,Y 334.056,Z 702.318,A -85,B 0,C 180,E1 22463.815,E2 22463.815} C_VEL
LIN {X 0,Y 327.365,Z 710.648,A -85,B 0,C 180,E1 22464.765,E2 22464.765} C_VEL
LIN {X 0,Y 319.158,Z 722.899,A -85,B 0,C 180,E1 22465.696,E2 22465.696} C_VEL
LIN {X 0,Y 315.646,Z 724.803,A -85,B 0,C 180,E1 22466.505,E2 22466.505} C_VEL
LIN {X 0,Y 309.25,Z 768.158,A -85,B 0,C 180,E1 22469.865,E2 22469.865} C_VEL
LIN {X 0,Y 303.205,Z 805.039,A -85,B 0,C 180,E1 22473.999,E2 22473.999} C_VEL
LIN {X 0,Y 297.74,Z 837.963,A -85,B 0,C 180,E1 22479.14,E2 22479.14} C_VEL
